					1:
						MEMCPY(ADR(MB_Type), ADR(DstBuf), MIN(MDP_Read.nCount, SIZEOF(MB_Type)) );
						MDP_Read.stMDP_DynAddr.nSubIdx		:= 2;

					2:
						MEMCPY(ADR(SerielNo), ADR(DstBuf), MIN(MDP_Read.nCount, SIZEOF(SerielNo)) );
						MDP_Read.stMDP_DynAddr.nSubIdx		:= 3;

					3:
						MEMCPY(ADR(ProdDate), ADR(DstBuf), MIN(MDP_Read.nCount, SIZEOF(ProdDate)) );
						MDP_Read.stMDP_DynAddr.nSubIdx		:= 4;

					4:
						MEMCPY(ADR(BootCount), ADR(DstBuf), SIZEOF(BootCount));
						MDP_Read.stMDP_DynAddr.nSubIdx		:= 5;

					5:
						MEMCPY(ADR(OpTime), ADR(DstBuf), SIZEOF(OpTime));
						MDP_Read.stMDP_DynAddr.nSubIdx		:= 6;

					6:
						MEMCPY(ADR(MinBoardTemp), ADR(DstBuf), SIZEOF(MinBoardTemp));
						MDP_Read.stMDP_DynAddr.nSubIdx		:= 7;

					7:
						MEMCPY(ADR(MaxBoardTemp), ADR(DstBuf), SIZEOF(MaxBoardTemp));
						MDP_Read.stMDP_DynAddr.nSubIdx		:= 8;

					8:
						MEMCPY(ADR(MinInputVolt), ADR(DstBuf), SIZEOF(MinInputVolt));
						MDP_Read.stMDP_DynAddr.nSubIdx		:= 9;

					9:
						MEMCPY(ADR(MaxInputVolt), ADR(DstBuf), SIZEOF(MaxInputVolt));
						MDP_Read.stMDP_DynAddr.nSubIdx		:= 10;

					10:
						MEMCPY(ADR(MB_Temp), ADR(DstBuf), SIZEOF(MB_Temp));
						MDP_Read.stMDP_DynAddr.nSubIdx		:= 0;
						MDP_Read.stMDP_DynAddr.nTableId		:= 4;
					END_CASE

				4:
					CASE MDP_Read.stMDP_DynAddr.nSubIdx OF
					0:
						MEMCPY(ADR(VoltCount), ADR(DstBuf), SIZEOF(VoltCount) );
						IF VoltCount > 0 THEN
							MDP_Read.stMDP_DynAddr.nSubIdx	:= 1;
						ELSE						
							state							:= 3;
						END_IF

					1..255:
						MEMCPY(ADR(VoltLocation[MDP_Read.stMDP_DynAddr.nSubIdx]), ADR(DstBuf), SIZEOF(VoltLocation[MIN_VOLTAGE]));
						MDP_Read.stMDP_DynAddr.nSubIdx	:= MDP_Read.stMDP_DynAddr.nSubIdx + 1;
						
						IF MDP_Read.stMDP_DynAddr.nSubIdx > VoltCount
						THEN
							MDP_Read.stMDP_DynAddr.nSubIdx	:= 1;
							MDP_Read.stMDP_DynAddr.nTableId	:= 5;
						END_IF
					END_CASE

				5:
					CASE MDP_Read.stMDP_DynAddr.nSubIdx OF
					1..255:
						MEMCPY(ADR(VoltageValue[MDP_Read.stMDP_DynAddr.nSubIdx]), ADR(DstBuf), SIZEOF(VoltageValue[MIN_VOLTAGE]));
						MDP_Read.stMDP_DynAddr.nSubIdx	:= MDP_Read.stMDP_DynAddr.nSubIdx + 1;
						
						IF MDP_Read.stMDP_DynAddr.nSubIdx > VoltCount
						THEN
							MDP_Read.stMDP_DynAddr.nSubIdx	:= 1;
							MDP_Read.stMDP_DynAddr.nTableId	:= 6;
						END_IF
					END_CASE

				6:
					CASE MDP_Read.stMDP_DynAddr.nSubIdx OF
					1..255:
						MEMCPY(ADR(VoltageNominal[MDP_Read.stMDP_DynAddr.nSubIdx]), ADR(DstBuf), SIZEOF(VoltageNominal[MIN_VOLTAGE]));
						MDP_Read.stMDP_DynAddr.nSubIdx	:= MDP_Read.stMDP_DynAddr.nSubIdx + 1;
						
						IF MDP_Read.stMDP_DynAddr.nSubIdx > VoltCount
						THEN
							state							:= 3;
						END_IF
					END_CASE
				END_CASE

				MDP_Read(
					stMDP_DynAddr	:= ,		(* address to request subindex Count of AdressList *)
					pDstBuf			:= ADR(DstBuf),
					cbDstBufLen		:= SIZEOF(DstBuf),
					bExecute		:= NOT MDP_Read.bBusy AND state = 2,
					tTimeout		:= Timeout,
					sAmsNetId		:= AmsNetId,
					bBusy			=> ,
					bError			=> ,
					nErrId			=> );
			END_IF
		END_IF

	3: //Start lesen der IPC Seriennummer 
		MDP_Read.stMDP_DynAddr.nArea						:= INT_TO_BYTE(eMDP_Area_DeviceArea);
		MDP_Read.stMDP_DynAddr.nModuleId					:= 16#9F;
		MDP_Read.stMDP_DynAddr.nTableId						:= 16#00;
		MDP_Read.stMDP_DynAddr.nSubIdx						:= 16#00;
		
		MDP_Read(
			stMDP_DynAddr	:= ,		(* address to request subindex Count of AdressList *)
			pDstBuf			:= ADR(IPC_SerielNo),
			cbDstBufLen		:= SIZEOF(IPC_SerielNo),
			bExecute		:= NOT MDP_Read.bBusy,
			tTimeout		:= Timeout,
			sAmsNetId		:= AmsNetId,
			bBusy			=> ,
			bError			=> ,
			nErrId			=> );	
			
		state												:= 4;	
	
	4:
		MDP_Read( pDstBuf	:= ADR(IPC_SerielNo), cbDstBufLen := SIZEOF(IPC_SerielNo));
		IF NOT MDP_Read.bBusy
		THEN
			IF MDP_Read.bError AND MDP_Read.bExecute
			THEN
				Busy										:= FALSE;
				Error										:= TRUE;
				SplitErrorId(
					nErrID		:= MDP_Read.nErrID,
					eErrGroup	=> ErrorGrp ,
					nErrCode	=> ErrorId);
				state										:= 99;	
			ELSE			                        		
				Busy										:= FALSE;
				Done										:= TRUE;
				state										:= 99;
			END_IF
			MDP_Read(bExecute := FALSE);
			
		END_IF

	99: ;

	ELSE
		;
	END_CASE


	(* reset state for next start *)
	IF NOT Execute
		AND state = 99
	THEN
		state												:= 0;
	END_IF

(****************************************************************************************************)

END_FUNCTION_BLOCK

// POUs/IpcDiag/MDP/InfoModuls/MDP_RaidSimple
{attribute 'no_check'}
FUNCTION_BLOCK MDP_RaidSimple  EXTENDS FbBase
VAR_OUTPUT CONSTANT
	MIN_DRIVE												:	INT := 1;
	MAX_DRIVE												:	INT := 4;
	                    									
//Cntr state            									
	CS_UNKNOWN												:	INT := 0;
	CS_GOOD													:	INT := 1;
	CS_FAILED												:	INT := 2; 
	CS_OFFLINE												:	INT := 3; 
	CS_POWER_OFF											:	INT := 4;
	                    									
//Cntr offline reason   									
	COR_NO_REASON											:	INT := 0;
	COR_INITIALIZING										:	INT := 1;
	COR_BUS_DEGRADED										:	INT := 2;
	COR_BUS_FAILURE											:	INT := 3;
	                    									
//Set state             									
	SS_OK													:	INT := 0;
	SS_DEGRADED												:	INT := 1;
	SS_REBUILDING											:	INT := 2;
	SS_FAILED												:	INT := 3;
	                    									
//Drive state		    									
	DS_OK													:	INT := 0;
	DS_REBUILDING											:	INT := 1;
	DS_FAILED 												:	INT := 2;
	DS_DEGRADED 											:	INT := 3;
END_VAR                 									
VAR_INPUT               									
	AmsNetId												: 	T_AmsNetId := '';	//AmsNetId as text
	Timeout													:	TIME := DEFAULT_ADS_TIMEOUT;	//Ads timeout
END_VAR                 									
VAR_OUTPUT              									
(* Raid Data *)         									
	CntrState												:	INT := CS_UNKNOWN;		//current controller state
	CntrOfflReason 											: 	INT := COR_NO_REASON;	//reason for controller offline
                        									
	SetType													:	USINT;					//type of RAID system
	SetState												:	INT := SS_OK;			
	SetInfo													:	USINT; (* 	If SetStatus = OK, THEN Info will be 0.
																					If SetStatus = DEGRADED, then Info will contain the failed drive index number.1
																					If SetStatus = REBUILDING, then Info will contain the percentage complete. The value will be in the range of 0 to 100 (0h to 64h).
																					If SetStatus == FAILED, then Info will be 0 or vendor specific. Since the failure modes could include drive or controller failures, Info may provide a vendor specific error code to indicate which component led to the failed status. *)
	CountDrives												:	UINT;
	DriveSTATE												:	ARRAY[MIN_DRIVE..MAX_DRIVE] OF INT; //current state of drive
	CountRAIDSets											:	UINT; 		//Count RAID sets
	ErrorGrp												:	E_MDP_ErrGroup := eMDP_Err_NoError;
END_VAR                 									
VAR                     									
	idx														:	INT := 1;
	MDP_ScanModules											:	FB_MDP_ScanModules := ( nModuleType 	:= eMDP_ModT_RAID , iModIdx		:= 0);
	MDP_Read												: 	FB_MDP_Read;
	SplitErrorId											:	FB_MDP_SplitErrorID ;
	DstBuf													:	ARRAY[0..4] OF BYTE;
END_VAR

(* Read RAID Information 						V1.0	*)
(* only for RAID set 1									*)
(* not more then MAX_DRIVES per RAID set				*)
(********************************************************)

(* Start Read *******************************************)
	IF Execute
		AND state = 0
	THEN
		CntrState											:= CS_UNKNOWN;
		CntrOfflReason 										:= COR_NO_REASON;
		SetType												:= 0;
		SetState											:= SS_OK;
		SetInfo												:= 0;
		CountDrives											:= 0;
		MEMSET(ADR(DriveSTATE),0,SIZEOF(DriveSTATE));   	
		CountRAIDSets										:= 0;
                                                        	
		Busy												:= TRUE;
		Done												:= FALSE;
		Error												:= FALSE;
		ErrorId												:= 0;
		ErrorGrp											:= eMDP_Err_NoError;
		MDP_Read(bExecute := FALSE);
		MDP_ScanModules(
			bExecute		:= FALSE,
			nModuleType		:= eMDP_ModT_RAID,
			iModIdx			:= 0,
			tTimeout		:= timeout,
			sAmsNetId		:= AmsNetId,
			bBusy			=> ,
			bError			=> ,
			nErrID			=> ,
			nDynModuleId	=> ,
			iModuleTypeCount=> ,
			iModuleCount	=> );
			
		MDP_ScanModules(bExecute:= TRUE);
		state												:= 1;
	ELSIF NOT Execute
		AND State = 99
	THEN
		state												:= 0;
		Busy												:= FALSE;
		Done												:= FALSE;
		Error												:= FALSE;
		ErrorId												:= 0;
		ErrorGrp											:= eMDP_Err_NoError;
	END_IF


	CASE state OF
	0:
		;
	1:
		MDP_ScanModules();
		IF NOT MDP_ScanModules.bBusy
		THEN
			IF MDP_ScanModules.bError
			THEN
				Busy										:= FALSE;
				Error										:= TRUE;
				SplitErrorId(
					nErrID		:= MDP_ScanModules.nErrID,
					eErrGroup	=> ErrorGrp ,
					nErrCode	=> ErrorId);
				state										:= 99;
				MDP_ScanModules(bExecute := FALSE);
			ELSE
				MDP_Read(bExecute := FALSE);
				MDP_Read.stMDP_DynAddr.nArea				:= 16#8;
				MDP_Read.stMDP_DynAddr.nModuleId			:= MDP_ScanModules.nDynModuleId;
				MDP_Read.stMDP_DynAddr.nTableId				:= 16#1;
				MDP_Read.stMDP_DynAddr.nSubIdx				:= 0;
				state										:= 2;
			END_IF

		END_IF

	2:
		MDP_Read( pDstBuf	:= ADR(DstBuf), cbDstBufLen := SIZEOF(DstBuf));
		IF NOT MDP_Read.bBusy
		THEN
			IF MDP_Read.bError AND MDP_Read.bExecute
			THEN
				IF MDP_Read.stMDP_DynAddr.nTableId = 16#2
					AND MDP_Read.stMDP_DynAddr.nSubIdx = 1
				THEN (* No RaidSystem found *)
					Busy									:= FALSE;
					Done									:= TRUE;
					state									:= 99;
				ELSE
					Busy									:= FALSE;
					Error									:= TRUE;
					SplitErrorId(
						nErrID		:= MDP_Read.nErrID,
						eErrGroup	=> ErrorGrp ,
						nErrCode	=> ErrorId);
				END_IF
				state										:= 99;
				MDP_Read(bExecute := FALSE);
			ELSE
				MDP_Read(bExecute := FALSE);
				CASE MDP_Read.stMDP_DynAddr.nTableId OF
				16#1: (* Controller Info *)
					CASE MDP_Read.stMDP_DynAddr.nSubIdx	OF
					0:
						MDP_Read.stMDP_DynAddr.nSubIdx		:= 1;

					1:
						MEMCPY(ADR(CntrState), ADR(DstBuf), SIZEOF(CntrState));
						MDP_Read.stMDP_DynAddr.nSubIdx		:= 2;

					2:
						MEMCPY(ADR(CntrOfflReason), ADR(DstBuf), SIZEOF(CntrOfflReason));
						MDP_Read.stMDP_DynAddr.nSubIdx		:= 0;
						MDP_Read.stMDP_DynAddr.nTableId		:= 16#2;
					END_CASE

				16#2: (* Raid Sets Type *)
					CASE MDP_Read.stMDP_DynAddr.nSubIdx	OF
					0:
						MEMCPY(ADR(CountRAIDSets), ADR(DstBuf), SIZEOF(CountRAIDSets));
						MDP_Read.stMDP_DynAddr.nSubIdx		:= 1;

					1:
						MEMCPY(ADR(SetType), ADR(DstBuf), SIZEOF(SetType));
						MDP_Read.stMDP_DynAddr.nSubIdx		:= 1;
						MDP_Read.stMDP_DynAddr.nTableId		:= 16#3;
					END_CASE

				16#3: (* RAID sets state and info *)
					CASE MDP_Read.stMDP_DynAddr.nSubIdx	OF
					1:
						MEMCPY(ADR(SetState), ADR(DstBuf[0]), 1);
						MEMCPY(ADR(SetInfo), ADR(DstBuf[1]), 1);
						MDP_Read.stMDP_DynAddr.nSubIdx		:= 0;
						MDP_Read.stMDP_DynAddr.nTableId		:= 16#A;
					END_CASE


				16#A: (* Drives state  *)
					CASE MDP_Read.stMDP_DynAddr.nSubIdx	OF
					0:
						MEMCPY(ADR(CountDrives), ADR(DstBuf), SIZEOF(CountDrives));
						MDP_Read.stMDP_DynAddr.nSubIdx		:= 1;

					1..255:
						MEMCPY(ADR(DriveSTATE), ADR(DstBuf), 1);
						MDP_Read.stMDP_DynAddr.nSubIdx	:= MDP_Read.stMDP_DynAddr.nSubIdx + 1;
						IF MDP_Read.stMDP_DynAddr.nSubIdx > CountDrives
							OR MDP_Read.stMDP_DynAddr.nSubIdx > MAX_DRIVE
						THEN
							Busy							:= FALSE;
							Done							:= TRUE;
							state							:= 99;
						END_IF

					END_CASE

				ELSE
					Busy									:= FALSE;
					Done									:= TRUE;
					state									:= 99;
				END_CASE

				MDP_Read(
					stMDP_DynAddr	:= ,(* address to request subindex Count of AdressList *)
					pDstBuf			:= ADR(DstBuf),
					cbDstBufLen		:= SIZEOF(DstBuf),
					bExecute		:= NOT MDP_Read.bBusy AND state = 2,
					tTimeout		:= Timeout,
					sAmsNetId		:= AmsNetId,
					bBusy			=> ,
					bError			=> ,
					nErrId			=> );
			END_IF
		END_IF

	99: ;

	ELSE
		;
	END_CASE

	(* reset state for next start *)
	IF NOT Execute
		AND state = 99
	THEN
		state												:= 0;
	END_IF

(****************************************************************************************************)

END_FUNCTION_BLOCK

// POUs/IpcDiag/MDP/InfoModuls/MDP_ReadModulList
{attribute 'no_check'}
FUNCTION_BLOCK MDP_ReadModulList EXTENDS FbBase
VAR_INPUT
	AmsNetId												: 	T_AmsNetId := '';	//AmsNetId as text
	Timeout													:	TIME := DEFAULT_ADS_TIMEOUT;	//Ads timeout
END_VAR                     								
VAR_OUTPUT                  								
	ModulCount												:	USINT;	//number of modules
	ModulType												:	ARRAY[0..255] OF E_MDP_ModuleType; //Index = Modul ID
	ErrorGrp												:	E_MDP_ErrGroup := eMDP_Err_NoError;
END_VAR                     								
VAR                         								
	MDP_Read												: 	FB_MDP_Read		:= (stMDP_DynAddr := (nArea := INT_TO_BYTE(eMDP_Area_DeviceArea), nModuleId := 16#02, nTableId := 16#00, nFlag := 16#00, nSubIdx := 16#00));
	SplitErrorId											:	FB_MDP_SplitErrorID;
	dwData													:	ARRAY [1..2] OF WORD;
END_VAR

(* Read list ob available moduls			V1.0	*)
(****************************************************)

(* Start read ************************************************)
	IF Execute
		AND state = 0
	THEN
		IF FALSE
		THEN (* Modultypen Liste *)
			MDP_Read.stMDP_DynAddr.nModuleId				:= 16#01;
		ELSE (* Modul ID Liste *)               			
			MDP_Read.stMDP_DynAddr.nModuleId				:= 16#02;
		END_IF                                  			
		MDP_Read.stMDP_DynAddr.nSubIdx						:= 0;
		MEMSET(ADR(ModulType),0,SIZEOF(ModulType));
		ModulCount											:= 0;
		Busy												:= TRUE;
		Done												:= FALSE;
		Error												:= FALSE;
		ErrorId												:= 0;
		ErrorGrp											:= eMDP_Err_NoError;
		
		MDP_Read(
			stMDP_DynAddr	:= ,		(* address to request subindex Count of AdressList *)
			pDstBuf			:= ADR(dwData),
			cbDstBufLen		:= SIZEOF(dwData),
			bExecute		:= FALSE,
			tTimeout		:= Timeout,
			sAmsNetId		:= AmsNetId,
			bBusy			=> ,
			bError			=> ,
			nErrId			=> );

		MDP_Read(bExecute	:= TRUE);
		state												:= 1;
	ELSIF NOT Execute
		AND State = 99
	THEN
		state												:= 0;
		Busy												:= FALSE;
		Done												:= FALSE;
		Error												:= FALSE;
		ErrorId												:= 0;
		ErrorGrp											:= eMDP_Err_NoError;
	END_IF


	CASE state OF
	0:
		;
	1:
		MDP_Read(pDstBuf := ADR(dwData), cbDstBufLen := SIZEOF(dwData));
		IF NOT MDP_Read.bBusy
		THEN
			IF MDP_Read.bError AND MDP_Read.bExecute
			THEN
				Busy										:= FALSE;
				Error										:= TRUE;
				SplitErrorId(
					nErrID		:= MDP_Read.nErrID,
					eErrGroup	=> ErrorGrp ,
					nErrCode	=> ErrorId);
				state										:= 99;
				MDP_Read(bExecute := FALSE);
			ELSE
				IF ModulCount = 0
				THEN (* Init Modul count *)
					ModulCount								:= WORD_TO_USINT(dwData[1]);
				ELSIF MDP_Read.stMDP_DynAddr.nSubIdx > 0
				THEN (* copy emlement dat					a *)
					ModulType[MDP_Read.stMDP_DynAddr.nSubIdx - 1] :=  dwData[2];					
				END_IF
				MDP_Read(bExecute := FALSE);
				MDP_Read.stMDP_DynAddr.nSubIdx:= MDP_Read.stMDP_DynAddr.nSubIdx + 1;
				IF MDP_Read.stMDP_DynAddr.nSubIdx > ModulCount
					OR MDP_Read.stMDP_DynAddr.nSubIdx > 255
				THEN
					Busy									:= FALSE;
					Done									:= TRUE;
					state									:= 99;
				ELSE
					MDP_Read(bExecute := TRUE,	pDstBuf	:= ADR(dwData), cbDstBufLen := SIZEOF(dwData));
				END_IF
			END_IF

		END_IF

	99: ;

	ELSE
		;
	END_CASE

	(* reset state for next start *)
	IF NOT Execute
		AND state = 99
	THEN
		state												:= 0;
	END_IF

(****************************************************************************************************)

END_FUNCTION_BLOCK

// POUs/IpcDiag/MDP/InfoModuls/MDP_SiliconDrives
{attribute 'no_check'}
FUNCTION_BLOCK MDP_SiliconDrives  EXTENDS FbBase
VAR_OUTPUT CONSTANT
	MIN_DRIVES												:	INT := 1;
	MAX_DRIVES												:	INT := 4;
END_VAR                 									
VAR_INPUT               									
	AmsNetId												: 	T_AmsNetId := '';	//AmsNetId as text
	Timeout													:	TIME := DEFAULT_ADS_TIMEOUT;	//Ads timeout
END_VAR                 									
VAR_OUTPUT              									
	TotEraseCounts											:  ARRAY[MIN_DRIVES..MAX_DRIVES] OF	T_LARGE_INTEGER;	//total number erase operations
	Usage													:	ARRAY[MIN_DRIVES..MAX_DRIVES] OF	UINT;	//usage of drive in %
	NoOfSpares												:	ARRAY[MIN_DRIVES..MAX_DRIVES] OF	UINT;	//number of partitions
	SparedUsed												:	ARRAY[MIN_DRIVES..MAX_DRIVES] OF	UINT;	//usage of partitions
	Count													:	INT; 	//number of drives
	NoSiliconDrives											:	BOOL := FALSE;	//should be TRUE if there is no SSD drive in use
	ErrorGrp												:	E_MDP_ErrGroup := eMDP_Err_NoError;
END_VAR
VAR
	idx														:	INT := 1;
	MDP_ScanModules											:	FB_MDP_ScanModules := ( nModuleType 	:= eMDP_ModT_SiliconDrive , iModIdx		:= 0);
	MDP_Read												: 	FB_MDP_ReadModuleContent;
	SplitErrorId											:	FB_MDP_SplitErrorID;
	DstBuf													:	ARRAY[0..8] OF BYTE;
END_VAR

	(* Read CPU Information 					V1.0	*)
	(****************************************************)

(* Start Read *******************************************************)
	IF Execute
		AND state = 0
	THEN
		MEMSET(ADR(TotEraseCounts),0,SIZEOF(TotEraseCounts));
		MEMSET(ADR(Usage),0,SIZEOF(Usage));
		MEMSET(ADR(NoOfSpares),0,SIZEOF(NoOfSpares));
		MEMSET(ADR(SparedUsed),0,SIZEOF(SparedUsed));
	
		NoSiliconDrives										:= FALSE;
		Count												:= 0;
		Busy												:= TRUE;
		Done												:= FALSE;
		Error												:= FALSE;
		ErrorId												:= 0;
		ErrorGrp											:= eMDP_Err_NoError;
		MDP_Read(bExecute := FALSE);
		MDP_ScanModules(
			bExecute		:= NOT MDP_ScanModules.bExecute,
			nModuleType		:= eMDP_ModT_SiliconDrive,
			iModIdx			:= 0,
			tTimeout		:= timeout,
			sAmsNetId		:= AmsNetId,
			bBusy			=> ,
			bError			=> ,
			nErrID			=> ,
			nDynModuleId	=> ,
			iModuleTypeCount=> ,
			iModuleCount	=> );
		MDP_ScanModules(bExecute := TRUE);
		
		state												:= 1;
	ELSIF NOT Execute
		AND State = 99
	THEN
		state												:= 0;
		Busy												:= FALSE;
		Done												:= FALSE;
		Error												:= FALSE;
		ErrorId												:= 0;
		ErrorGrp											:= eMDP_Err_NoError;
	END_IF


	CASE state OF
	0:
		;
	1:
		MDP_ScanModules();
		IF NOT MDP_ScanModules.bBusy
		THEN
			IF MDP_ScanModules.bError
			THEN
				IF MDP_ScanModules.nErrID = 16#EC800002
				THEN
					Busy									:= FALSE;
					Done									:= TRUE;
					NoSiliconDrives							:= TRUE;
				ELSE

					Busy									:= FALSE;
					Error									:= TRUE;
					SplitErrorId(
						nErrID		:= MDP_ScanModules.nErrID,
						eErrGroup	=> ErrorGrp ,
						nErrCode	=> ErrorId);
				END_IF
				state										:= 99;
				MDP_ScanModules(bExecute := FALSE);
			ELSE
				Count										:= MDP_ScanModules.iModuleTypeCount;
				MDP_Read.stMDP_DynAddr.nArea				:= 16#8;
				MDP_Read.stMDP_DynAddr.nModuleId			:= MDP_ScanModules.nDynModuleId;
				MDP_Read.stMDP_DynAddr.nSubIdx				:= 0;
				MDP_Read.stMDP_DynAddr.nTableId				:= 1;
				MDP_Read(bExecute := FALSE);
				idx											:= 1;
				
				IF Count <= 0
				THEN
					Busy									:= FALSE;
					Done									:= TRUE;
					state									:= 99;
				ELSE
					state									:= 2;
				END_IF
			END_IF

		END_IF

	2:
		MDP_Read( pDstBuf:= ADR(DstBuf), cbDstBufLen:= SIZEOF(DstBuf));
		IF NOT MDP_Read.bBusy
		THEN
			IF MDP_Read.bError AND MDP_Read.bExecute
			THEN
				Busy										:= FALSE;
				Error										:= TRUE;
				SplitErrorId(
					nErrID		:= MDP_Read.nErrID,
					eErrGroup	=> ErrorGrp ,
					nErrCode	=> ErrorId);
				state										:= 99;
				MDP_Read(bExecute := FALSE);
			ELSE
				MDP_Read(bExecute := FALSE);
				CASE MDP_Read.stMDP_DynAddr.nSubIdx OF
				0:
					MDP_Read.stMDP_DynAddr.nSubIdx			:= 1;

				1:
					MEMCPY(ADR(TotEraseCounts[idx]), ADR(DstBuf), MIN(MDP_Read.nCount, SIZEOF(TotEraseCounts[MIN_DRIVES])));
					MDP_Read.stMDP_DynAddr.nSubIdx			:= 2;

				2:
					MEMCPY(ADR(Usage[idx]), ADR(DstBuf), SIZEOF(Usage[MIN_DRIVES]));
					MDP_Read.stMDP_DynAddr.nSubIdx			:= 3;

				3:
					MEMCPY(ADR(NoOfSpares[idx]), ADR(DstBuf), SIZEOF(NoOfSpares[MIN_DRIVES]));
					MDP_Read.stMDP_DynAddr.nSubIdx			:= 4;

				4:
					MEMCPY(ADR(SparedUsed[idx]), ADR(DstBuf), SIZEOF(SparedUsed[MIN_DRIVES]));
					MDP_Read.stMDP_DynAddr.nModuleId		:= MDP_Read.stMDP_DynAddr.nModuleId + 1;
					idx										:= idx + 1;
					MDP_Read.stMDP_DynAddr.nSubIdx			:= 1;
					IF idx > Count
						OR idx > MAX_DRIVES
					THEN
						Busy								:= FALSE;
						Done								:= TRUE;
						state								:= 99;
					END_IF
				END_CASE

				MDP_Read(
					stMDP_DynAddr	:= ,		(* address to request subindex Count of AdressList *)
					pDstBuf			:= ADR(DstBuf),
					cbDstBufLen		:= SIZEOF(DstBuf),
					bExecute		:= NOT MDP_Read.bBusy AND state = 2,
					tTimeout		:= Timeout,
					sAmsNetId		:= AmsNetId,
					bBusy			=> ,
					bError			=> ,
					nErrId			=> );

			END_IF
		END_IF

	99: ;

	ELSE
		;
	END_CASE

	(* reset state for next start *)
	IF NOT Execute
		AND state = 99
	THEN
		state												:= 0;
	END_IF

(****************************************************************************************************)

END_FUNCTION_BLOCK

// POUs/IpcDiag/MDP/InfoModuls/MDP_UPS
{attribute 'no_check'}
FUNCTION_BLOCK MDP_UPS EXTENDS FbBase
VAR_OUTPUT CONSTANT
(* Battery Power Status *)
	PS_UNKNOWN												:	INT := 0;
	PS_ONLINE												:	INT := 1;
	PS_ONBATTERIES											:	INT := 2;
	                    									
(* Com Status *)        									
	CS_UNKNOWN												:	INT := 0;
	CS_OK													:	INT := 1;
	CS_ERROR												:	INT := 2;

(* Battery Power Status *)
	BS_UNKNOWN												:	INT := 0;
	BS_OK													:	INT := 1;
	BS_CHANGE_BATTERY										:	INT := 2;
	
END_VAR
VAR_INPUT
	AmsNetId												: 	T_AmsNetId := '';	//AmsNetId
	Timeout													:	TIME := DEFAULT_ADS_TIMEOUT;	//Ads timeout
END_VAR
VAR_OUTPUT
(* UPS Data *)              								
	Model													:	STRING(30);	//model name
	VendorName												:	STRING(30);	//vendor name
	PowerStatus												:	INT := PS_UNKNOWN;
	ComStatus												:	INT := CS_UNKNOWN;
	BatteryStatus											:	INT := BS_UNKNOWN;
	BatteryCapacity											:	USINT; 		//in %
	BatteryRuntime											:	UDINT; 		//in sec
	PersPowerFailCounter									:	BOOL;		//TRUE when persistent power fail counter is activated
	PowerFailCounter										:	UDINT;		//number of power fails
	FanError												:	BOOL;		//Fan has error
	NoBattery												:	BOOL;		//No battery connected
	ErrorGrp												:	E_MDP_ErrGroup := eMDP_Err_NoError;

END_VAR                     								
VAR                         								
	idx														:	INT := 1;
	MDP_ScanModules											:	FB_MDP_ScanModules := ( nModuleType 	:= eMDP_ModT_UPS , iModIdx		:= 0);
	MDP_Read												: 	FB_MDP_Read;
	SplitErrorId											:	FB_MDP_SplitErrorID;
	DstBuf													:	ARRAY[0..31] OF BYTE;
END_VAR

	(* Read UPS Information 							V1.0	*)
	(***************************************************)

(* Start Read *******************************************************)
	IF Execute
		AND state = 0
	THEN
		Model												:= '';
		VendorName											:= '';
		PowerStatus											:= PS_UNKNOWN;
		ComStatus											:=	CS_UNKNOWN;
		BatteryStatus										:=	BS_UNKNOWN;
		BatteryCapacity										:= 0;
		BatteryRuntime										:= 0;
		PowerFailCounter									:= 0;
		PersPowerFailCounter								:= FALSE;
		FanError											:= FALSE;
		NoBattery											:= FALSE;
		Busy												:= TRUE;
		Done												:= FALSE;
		Error												:= FALSE;
		ErrorId												:= 0;
		ErrorGrp											:= eMDP_Err_NoError;
		MDP_Read(bExecute := FALSE);
		MDP_ScanModules(
			bExecute		:= NOT MDP_ScanModules.bExecute,
			nModuleType		:= eMDP_ModT_UPS,
			iModIdx			:= 0,
			tTimeout		:= timeout,
			sAmsNetId		:= AmsNetId,
			bBusy			=> ,
			bError			=> ,
			nErrID			=> ,
			nDynModuleId	=> ,
			iModuleTypeCount=> ,
			iModuleCount	=> );
			
		MDP_ScanModules(bExecute := TRUE);
		
		state												:= 1;
	ELSIF NOT Execute
		AND State = 99
	THEN
		state												:= 0;
		Busy												:= FALSE;
		Done												:= FALSE;
		Error												:= FALSE;
		ErrorId												:= 0;
		ErrorGrp											:= eMDP_Err_NoError;
	END_IF


	CASE state OF
	0:
		;
	1:
		MDP_ScanModules();
		IF NOT MDP_ScanModules.bBusy
		THEN
			IF MDP_ScanModules.bError
			THEN
				Busy										:= FALSE;
				Error										:= TRUE;
				SplitErrorId(
					nErrID		:= MDP_ScanModules.nErrID,
					eErrGroup	=> ErrorGrp ,
					nErrCode	=> ErrorId);
				state										:= 99;
				MDP_ScanModules(bExecute := FALSE);
			ELSE
				MDP_Read(bExecute := FALSE);
				MDP_Read.stMDP_DynAddr.nArea				:= 16#8;
				MDP_Read.stMDP_DynAddr.nModuleId			:= MDP_ScanModules.nDynModuleId;
				MDP_Read.stMDP_DynAddr.nTableId				:= 1;
				MDP_Read.stMDP_DynAddr.nSubIdx				:= 0;
				state										:= 2;
			END_IF

		END_IF

	2:
		MDP_Read( pDstBuf	:= ADR(DstBuf), cbDstBufLen := SIZEOF(DstBuf));
		IF NOT MDP_Read.bBusy
		THEN
			IF MDP_Read.bError AND MDP_Read.bExecute
			THEN
				Busy										:= FALSE;
				Error										:= TRUE;
				SplitErrorId(
					nErrID		:= MDP_Read.nErrID,
					eErrGroup	=> ErrorGrp ,
					nErrCode	=> ErrorId);
				state										:= 99;
				MDP_Read(bExecute := FALSE);
			ELSE
				MDP_Read(bExecute := FALSE);
				CASE MDP_Read.stMDP_DynAddr.nSubIdx	OF
				0:
					MDP_Read.stMDP_DynAddr.nSubIdx			:= 1;

				1:
					MEMCPY(ADR(Model), ADR(DstBuf), SIZEOF(Model) - 1);
					MDP_Read.stMDP_DynAddr.nSubIdx			:= 2;

				2:
					MEMCPY(ADR(VendorName), ADR(DstBuf), SIZEOF(VendorName) - 1);
					MDP_Read.stMDP_DynAddr.nSubIdx			:= 7;

				7:
					MEMCPY(ADR(PowerStatus), ADR(DstBuf), 1);
					MDP_Read.stMDP_DynAddr.nSubIdx			:= 8;

				8:
					MEMCPY(ADR(ComStatus), ADR(DstBuf), 1);
					MDP_Read.stMDP_DynAddr.nSubIdx			:= 9;

				9:
					MEMCPY(ADR(BatteryStatus), ADR(DstBuf), 1);
					MDP_Read.stMDP_DynAddr.nSubIdx			:= 10;

				10:
					MEMCPY(ADR(BatteryCapacity), ADR(DstBuf), SIZEOF(BatteryCapacity));
					MDP_Read.stMDP_DynAddr.nSubIdx			:= 11;

				11:
					MEMCPY(ADR(BatteryRuntime), ADR(DstBuf), SIZEOF(BatteryRuntime));
					MDP_Read.stMDP_DynAddr.nSubIdx			:= 12;

				12:
					MEMCPY(ADR(PersPowerFailCounter), ADR(DstBuf), SIZEOF(PersPowerFailCounter));
					MDP_Read.stMDP_DynAddr.nSubIdx			:= 13;

				13:
					MEMCPY(ADR(PowerFailCounter), ADR(DstBuf), SIZEOF(PowerFailCounter));
					MDP_Read.stMDP_DynAddr.nSubIdx			:= 14;

				14:
					MEMCPY(ADR(FanError), ADR(DstBuf), SIZEOF(FanError));
					MDP_Read.stMDP_DynAddr.nSubIdx			:= 15;

				15:
					MEMCPY(ADR(NoBattery), ADR(DstBuf), SIZEOF(NoBattery));
					Busy									:= FALSE;
					Done									:= TRUE;
					state									:= 99;
                                                        	
				ELSE                                    	
					Busy									:= FALSE;
					Done									:= TRUE;
					state									:= 99;
				END_CASE

				MDP_Read(
					stMDP_DynAddr	:= ,(* address to request subindex Count of AdressList *)
					pDstBuf			:= ADR(DstBuf),
					cbDstBufLen		:= SIZEOF(DstBuf),
					bExecute		:= NOT MDP_Read.bBusy AND state = 2,
					tTimeout		:= Timeout,
					sAmsNetId		:= AmsNetId,
					bBusy			=> ,
					bError			=> ,
					nErrId			=> );
			END_IF
		END_IF

	99: ;

	ELSE
		;
	END_CASE

	(* reset state for next start *)
	IF NOT Execute
		AND state = 99
	THEN
		state												:= 0;
	END_IF

(****************************************************************************************************)

END_FUNCTION_BLOCK

// POUs/IpcDiag/MDP/MDP_Info
{attribute 'no_check'}
//Wrapper for available MDP_xxxx FBs of the lib, based on Beckhoff MDP - invalid values are reported via EventLogger 
//based on Tc2_MDP.lib - please see Beckhoff documentation for further information about Tc2_MDP.lib (IPC diagnostics)
FUNCTION_BLOCK MDP_Info EXTENDS FbBase
VAR_OUTPUT CONSTANT
	FNC_READ_ALL											:	INT := 0;
	FNC_READ_MOD_LIST										:	INT := 1;
	FNC_READ_MB												:	INT := 2;
	FNC_READ_CPU											:	INT := 3;
	FNC_READ_FAN											:	INT := 4;
	FNC_READ_SD												:	INT := 5;
	FNC_READ_RAID											:	INT := 6;
	FNC_READ_UPS											:	INT := 7;
END_VAR                 									
VAR_INPUT               									
	AmsNetId												: 	T_AmsNetId := '';	//AmsNetId as text
	Timeout													:	TIME := DEFAULT_ADS_TIMEOUT; //Ads timeout
	Fnc														:	INT (FNC_READ_ALL..FNC_READ_UPS) := FNC_READ_ALL; //select function to be read
(* Components *)            								
	ModList													:	MDP_ReadModulList;	//see content in FB
	MB														:	MDP_Mainboard;		//see content in FB
	CPU														:	MDP_CPU;			//see content in FB
	FAN														:	MDP_Fan;			//see content in FB
	SD														:	MDP_SiliconDrives;	//see content in FB
	RAID													:	MDP_RaidSimple;		//see content in FB
	UPS														:	MDP_UPS;			//see content in FB
END_VAR                     								
VAR_OUTPUT                  								
	TotalCycleTime											:	TIME;	//Cylce time to execute function block with mode read all        
	ErrorGrp												:	E_MDP_ErrGroup;
	ErrorFnc												:	STRING(15);
END_VAR
VAR
	MemFnc													:	INT;
	MemExecute												:	BOOL;
	MemErrorFnc												:	STRING(15);
	MemErrorid												:	UDINT;
	MemErrorGrp												:	E_MDP_ErrGroup;
	MemTimeStartCycle										:	TIME;
END_VAR

	(* Execute all available MDP_xxxxx fb 			*)
	(************************************************)

(* Sequence ********************************************)
	IF Execute
		AND state = 0
	THEN
		ReadAll(Execute	:= Execute);
	ELSIF state <> 0
	THEN
		ReadAll(Execute	:= Execute);
	END_IF

(*****************************************************************************)

METHOD PUBLIC readAll : BOOL //Return value = TRUE if busy;
VAR_INPUT
	Execute													:	BOOL;
END_VAR
	THIS^.Execute											:= Execute;

	IF Execute
		AND State = 0
	THEN
		MemFnc												:= Fnc;
		CASE Fnc OF                                     	
		FNC_READ_MOD_LIST:		state						:= 10;
		FNC_READ_MB:			state						:= 20;
		FNC_READ_CPU:			state						:= 30;
		FNC_READ_FAN:			state						:= 40;
		FNC_READ_SD:			state						:= 50;
		FNC_READ_RAID:	 		state						:= 60;
		FNC_READ_UPS:	 		state						:= 70;
		ELSE (* Read All *)
			MemFnc											:= FNC_READ_ALL;
			state											:= 10;
		END_CASE
		MemTimeStartCycle									:= TIME();
		Busy												:= TRUE;
		Done												:= FALSE;
		Error												:= FALSE;
		Errorid												:= 0;
		ErrorFnc											:= '';
		ErrorGrp											:= eMDP_Err_NoError;
		MemExecute											:= FALSE;
		MemErrorid											:= 0;
		MemErrorFnc											:= '';
		MemErrorGrp											:= eMDP_Err_NoError;
	ELSIF NOT Execute
		AND State = 99
	THEN
		Busy												:= FALSE;
		Done												:= FALSE;
		Error												:= FALSE;
		Errorid												:= 0;
		ErrorFnc											:= '';
		ErrorGrp											:= eMDP_Err_NoError;
		MemExecute											:= FALSE;
		MemErrorid											:= 0;
		MemErrorFnc											:= '';
		MemErrorGrp											:= eMDP_Err_NoError;
		ReadModList(FALSE);     						
		ReadMB(FALSE);
		ReadCPU(FALSE);
		ReadFAN(FALSE);
		ReadSD(FALSE);
		ReadRaid(FALSE);
	END_IF

	CASE state OF
	10:

		MemExecute											:= TRUE;
		ReadModList(MemExecute);
		IF NOT ModList.Busy
		THEN
			IF MemFnc = FNC_READ_ALL
			THEN
				IF Error AND MemErrorid = 0 
				THEN
					MemErrorId								:= Errorid; 
					MemErrorFnc 							:= CONCAT('ReadModList Fnc:',TO_STRING(FNC_READ_MOD_LIST)); 
					MemErrorGrp 							:= ErrorGrp;
				END_IF              						
				Busy										:= TRUE;
				Done										:= FALSE;
				Error										:= FALSE;
				Errorid										:= 0;
				ErrorGrp									:= eMDP_Err_NoError;
				state										:= 20;
			ELSE                    						
				state										:= 99;
			END_IF
		END_IF

	20:
		MemExecute											:= TRUE;
		ReadMB(MemExecute);
		IF NOT MB.Busy
		THEN
			IF MemFnc = FNC_READ_ALL
			THEN
				IF Error AND MemErrorid = 0 
				THEN
					MemErrorId								:= Errorid; 
					MemErrorFnc 							:= CONCAT('ReadMB Fnc: ',TO_STRING(FNC_READ_MB));  
					MemErrorGrp 							:= ErrorGrp;
				END_IF              						
				Busy										:= TRUE;
				Done										:= FALSE;
				Error										:= FALSE;
				Errorid										:= 0;
				ErrorGrp									:= eMDP_Err_NoError;
				state										:= 30;
			ELSE                    						
				state										:= 99;
			END_IF                  	
		END_IF

	30:
		MemExecute											:= TRUE;
		ReadCPU(MemExecute);
		IF NOT CPU.Busy
		THEN
			IF MemFnc = FNC_READ_ALL
			THEN
				IF Error AND MemErrorid = 0 THEN
					MemErrorId								:= Errorid; 
					MemErrorFnc 							:= CONCAT('ReadCPU Fnc: ',TO_STRING(FNC_READ_CPU));  
					MemErrorGrp 							:= ErrorGrp;
				END_IF              						
				Busy										:= TRUE;
				Done										:= FALSE;
				Error										:= FALSE;
				Errorid										:= 0;
				ErrorGrp									:= eMDP_Err_NoError;
				state										:= 40;
			ELSE                    						
				state										:= 99;
			END_IF
		END_IF

	40:
		MemExecute											:= TRUE;
		ReadFan(MemExecute);
		IF NOT Fan.Busy
		THEN
			IF MemFnc = FNC_READ_ALL
			THEN
				IF Error AND MemErrorid = 0 
				THEN
					MemErrorId								:= Errorid; 
					MemErrorFnc 							:= CONCAT('ReadFan Fnc: ',TO_STRING(FNC_READ_FAN));  
					MemErrorGrp 							:= ErrorGrp;
				END_IF              						
				Busy										:= TRUE;
				Done										:= FALSE;
				Error										:= FALSE;
				Errorid										:= 0;
				ErrorGrp									:= eMDP_Err_NoError;
				state										:= 50;
			ELSE                    						
				state										:= 99;
			END_IF
		END_IF

	50:
		MemExecute											:= TRUE;		
		ReadSD(MemExecute);
		
		IF NOT SD.Busy
		THEN
			IF MemFnc = FNC_READ_ALL
			THEN
				IF Error AND MemErrorid = 0 
				THEN				
					MemErrorId								:= Errorid; 
					MemErrorFnc 							:= CONCAT('ReadSD Fnc: ',TO_STRING(FNC_READ_SD)); 
					MemErrorGrp 							:= ErrorGrp;
				END_IF              						
				Busy										:= TRUE;
				Done										:= FALSE;
				Error										:= FALSE;
				Errorid										:= 0;
				ErrorGrp									:= eMDP_Err_NoError;
				state										:= 60;
			ELSE                    						
				state										:= 99;
			END_IF                  	
		END_IF

	60:
		MemExecute											:= TRUE;
		ReadRaid(MemExecute);
		IF NOT Raid.Busy
		THEN
			IF MemFnc = FNC_READ_ALL
			THEN
				IF Error AND MemErrorid = 0 
				THEN
					MemErrorId								:= Errorid; 
					MemErrorFnc 							:= CONCAT('ReadRaid Fnc: ',TO_STRING(FNC_READ_RAID));
					MemErrorGrp 							:= ErrorGrp;
				END_IF              						
				Busy										:= TRUE;
				Done										:= FALSE;
				Error										:= FALSE;
				Errorid										:= 0;
				ErrorGrp									:= eMDP_Err_NoError;
				state										:= 70;
			ELSE                    						
				state										:= 99;
			END_IF
		END_IF

	70:
		MemExecute											:= TRUE;
		ReadUPS(MemExecute);
		IF NOT UPS.Busy
		THEN
			IF TRUE
			THEN
				IF Error AND MemErrorid = 0 
				THEN
					MemErrorId								:= Errorid; 
					MemErrorFnc 							:= CONCAT('ReadUPS Fnc: ',TO_STRING(FNC_READ_UPS));
					MemErrorGrp 							:= ErrorGrp;
				END_IF
				Busy										:= FALSE;
				Done										:= MemErrorId = 0;
				Error										:= MemErrorId <> 0;
				Errorid										:= MemErrorid;
				ErrorFnc									:= MemErrorFnc;
				ErrorGrp									:= MemErrorGrp;
				state										:= 99;
			ELSE                    						
				state										:= 99;
			END_IF
		END_IF

	99:;
	
	END_CASE

	IF state = 99
	THEN
		TotalCycleTime	 									:= TIME() - MemTimeStartCycle;
		IF NOT Execute
		THEN
			state											:= 0;
			ReadModList(FALSE);         					
			ReadMB(FALSE);              					
			ReadCPU(FALSE);             					
			ReadFAN(FALSE);             					
			ReadSD(FALSE);              					
			ReadRaid(FALSE);            					
			ReadUPS(FALSE);             	
		END_IF                          	
	END_IF                              	
	                                    	
	ReadAll													:= Busy;

(***********************************************************************************)
END_METHOD

METHOD PUBLIC readCPU : BOOL //Return value = TRUE if busy
VAR_INPUT
	Execute													:	BOOL;
END_VAR
THIS^.Execute												:= Execute;

CPU(
	Execute				:= MemExecute OR Execute,
	AmsNetId			:= AmsNetId,
	Timeout				:= Timeout,
	MIN_CPU				=> ,
	MAX_CPU				=> ,
	Busy				=> Busy,
	Done				=> Done,
	Error				=> Error,
	ErrorId				=> Errorid,
	ErrorGrp 			=> ErrorGrp,
	Frequency			=> ,
	Usage				=> ,
	Temperature			=> ,
	AverageFrequency	=> ,
	AverageUsage		=> ,
	AverageTemperature	=> ,
	Count				=> );

MemExecute 													:= FALSE;
	        												
ReadCPU														:= Busy;
END_METHOD

METHOD PUBLIC readFan : BOOL //Return value = TRUE if busy
VAR_INPUT
	Execute													:	BOOL;
END_VAR
THIS^.Execute												:= Execute;

FAN(
	Execute		:= MemExecute OR Execute,
	AmsNetId	:= AmsNetid,
	Timeout		:= Timeout,
	MIN_FAN		=> ,
	MAX_FAN		=> ,
	Busy		=> Busy,
	Done		=> Done,
	Error		=> Error,
	ErrorId		=> ErrorId,
	ErrorGrp 	=> ErrorGrp,
	Speed		=> ,
	Count		=> );

MemExecute 													:= FALSE;
           												
ReadFan														:= Busy;
END_METHOD

METHOD PUBLIC readMB : BOOL //Return value = TRUE if busy
VAR_INPUT
	Execute													:	BOOL;
END_VAR
THIS^.Execute												:= Execute;

MB(
	Execute			:= MemExecute OR Execute,
	AmsNetId		:= AmsNetId,
	Timeout			:= Timeout,
	MIN_VOLTAGE		=> ,
	MAX_VOLTAGE		=> ,
	Busy			=> Busy,
	Done			=> Done,
	Error			=> Error,
	ErrorId			=> ErrorId,
	ErrorGrp		=> Errorgrp,
	MB_Type			=> ,
	SerielNo		=> ,
	ProdDate		=> ,
	BootCount		=> ,
	OpTime			=> ,
	MinBoardTemp	=> ,
	MaxBoardTemp	=> ,
	MinInputVolt	=> ,
	MaxInputVolt	=> ,
	MB_Temp			=> ,
	VoltLocation	=> ,
	VoltageValue	=> ,
	VoltageNominal	=> ,
	VoltCount		=> );

MemExecute 													:= FALSE;
            												
ReadMB														:= Busy;
END_METHOD

METHOD PUBLIC readModList : BOOL //Return value = TRUE if busy
VAR_INPUT
	Execute													:	BOOL;
END_VAR
THIS^.Execute												:= Execute;

ModList(
	Execute		:= MemExecute OR Execute,
	AmsNetId	:= AmsNetId,
	Timeout		:= Timeout,
	Busy		=> Busy,
	Done		=> done,
	Error		=> Error,
	ErrorId		=> ErrorId,
	ErrorGrp 	=> ErrorGrp );

MemExecute 													:= FALSE;
            												
ReadModList													:= Busy;
END_METHOD

METHOD PUBLIC readRaid : BOOL //Return value = TRUE if busy
VAR_INPUT
	Execute													: BOOL;
END_VAR
THIS^.Execute												:= Execute;

RAID(
	Execute			:= Execute OR MemExecute,
	AmsNetId		:= AmsNetId,
	Timeout			:= timeout,
	MIN_DRIVE		=> ,
	MAX_DRIVE		=> ,
	Busy			=> Busy,
	Done			=> done,
	Error			=> Error,
	ErrorId			=> ErrorId,
	ErrorGrp 		=> ErrorGrp,
	CntrState		=> ,
	CntrOfflReason	=> ,
	SetType			=> ,
	SetState		=> ,
	SetInfo			=> ,
	CountDrives		=> ,
	DriveSTATE		=> ,
	CountRAIDSets	=> );

MemExecute 													:= FALSE;
                											
ReadRaid													:= Busy;
END_METHOD

METHOD PUBLIC readSD : BOOL //Return value = TRUE if busy
VAR_INPUT
	Execute		:	BOOL;
END_VAR
THIS^.Execute												:= Execute;

SD(
	Execute			:= MemExecute OR Execute,
	AmsNetId		:= AmsNetid,
	Timeout			:= timeout,
	MIN_DRIVES		=> ,
	MAX_DRIVES		=> ,
	Busy			=> Busy,
	Done			=> Done,
	Error			=> Error,
	ErrorId			=> Errorid,
	ErrorGrp 		=> ErrorGrp,
	TotEraseCounts	=> ,
	Usage			=> ,
	NoOfSpares		=> ,
	SparedUsed		=> ,
	Count			=> );

MemExecute	 												:= FALSE;
                											
ReadSD														:= Busy;
END_METHOD

METHOD PUBLIC readUPS : Bool //Return value = TRUE if busy
VAR_INPUT
	Execute		:	BOOL;
END_VAR
THIS^.Execute												:= Execute;

UPS(
	Execute					:= MemExecute OR Execute,
	AmsNetId				:= AmsNetid,
	Timeout					:= timeout,
	Busy					=> Busy,
	Done					=> Done,
	Error					=> Error,
	ErrorId					=> Errorid,
	ErrorGrp				=> ErrorGrp,
	Model					=> ,
	VendorName				=> ,
	PowerStatus				=> ,
	ComStatus				=> ,
	BatteryStatus			=> ,
	BatteryCapacity			=> ,
	BatteryRuntime			=> ,
	PersPowerFailCounter	=> ,
	PowerFailCounter		=> ,
	FanError				=> ,
	NoBattery				=> );

MemExecute 													:= FALSE;
ReadUPS														:= Busy;
END_METHOD

END_FUNCTION_BLOCK

// POUs/IpcDiag/MDP/MDP_IpcDiag
{attribute 'no_check'}
//General IPC diagnosis based on Beckhoff MDP - invalid values are reported via EventLogger 
//based on Tc2_MDP.lib - please see Beckhoff documentation for further information about Tc2_MDP.lib (IPC diagnostics)
//EventHandlingGrp10 instance used inside
//Info:
// 0x   	a    	nn   	x   
// 0x   	8   	03   	1   
// a 	= Area Code (e.g. 8 = Configuration Area) 
// nn 	= Modul-ID (e.g. dynamic modul id from list F020) 
// x	= Tabel id (e.g. 1 = Table 0x8nn1 - NIC Properties at area code 8) 
FUNCTION_BLOCK MDP_IpcDiag
VAR CONSTANT
	MIN_CPU													:	INT := 1;
	MAX_CPU													:	INT := 4;
	                    									
	MIN_FAN													:	INT := 1;
	MAX_FAN													:	INT := 4;
	                    									
	MIN_VOLTAGE												:	INT := 1;
	MAX_VOLTAGE												:	INT := 8;		
END_VAR                 									
VAR_INPUT               									
	Enable													:	BOOL := FALSE;	//FB will be processed as long as enable is TRUE 
	CycleTime												:	TIME := T#100MS; //Delay between ads call to read a single value 
	AmsNetId												: 	T_AmsNetId := ''; //Ams net Id
	Timeout													: 	TIME := DEFAULT_ADS_TIMEOUT; //Ads timeout
{attribute 'displaymode':='bin'}
	FanMask													:	BYTE := 2#0000_0011; //Installed fans inside the PC 
	
//Threshold values 	    									
	MinSpeedFan												:	INT := 2500; 	//rpm
	MaxTempMB												:	INT := 85; 		//°C
	MaxTempCPU												:	INT := 100; 	//°C
	TempWarningThreshold									:	INT := 10; 		//°C
	VoltageFactor											:	LREAL := 0.7; 	//% of nominal voltage before an error occurs
END_VAR                 									
VAR_OUTPUT              										                									
	MB_Temp													:	INT; //Motherboard temp with one decimal digit  
	Voltage_Count											:	INT := 0; //count of voltage measurement points with one decimal digit 
	MB_NominalVoltage										:	ARRAY[MIN_VOLTAGE..MAX_VOLTAGE] OF INT; //in mV
	MB_Voltage												:	ARRAY[MIN_VOLTAGE..MAX_VOLTAGE] OF INT;  //in mV
	CPU_Count												:	INT := 0; //Readed number of CPUs
	CPU_Temp												:	ARRAY[MIN_CPU..MAX_CPU] OF INT; //cpu temperatur with one decimal digit
	FAN_Count												:	INT := 0; //Number of FANs in config. Note, the number may be two where only the second fan is p
	FAN_Speed												:	ARRAY[MIN_FAN..MAX_FAN] OF INT; //in rpm for each available fan
	OsImage													:	STRING; //Image version 
	ExecutionTime											:	TIME; 	//Cylce time to execute function block        
	Busy													:	BOOL;	//Busy is TRUE at the rising edge of Enable and stays TRUE as long as the FB is performing any action. 
	Valid													:	BOOL;	//data valid
	Error													:	BOOL;	//Rising edge of Error informs that an error occurred during the execution of the Function Block 
{attribute 'displaymode':='hex'}
	ErrorId													:	UDINT;	//Error identification - see documentation about IPC diagnostic for further detailed informantion 
	ErrorGrp												:	E_MDP_ErrGroup := eMDP_Err_NoError; //MDP Error code - see Beckhoff documentation MDP for further informantion
END_VAR	
VAR
(* cache variables ************************************************************)
	state													:	INT := 0;
	
	dwData													:	ARRAY [1..2] OF WORD;
	                    									
	MemLen													:	BYTE := 0;
	MemModIdMB												:	BYTE;
	MemModIdCPU												:	ARRAY[MIN_CPU..MAX_CPU] OF BYTE;
	MemModIdFan												:	ARRAY[MIN_FAN..MAX_FAN] OF BYTE;
	MEmModIdUPS												:	BYTE;
	MemMBSubIdxVoltage										:	ARRAY[MIN_VOLTAGE..MAX_VOLTAGE] OF BYTE;
	MemTimeStartCycle										:	TIME;
	MemErrState												:	INT := 0;
	
(* timer ***************************************************************************)
	TON_Cycle												:	TON;
	
(* function-blocks *****************************************************************)
	MDP_Read												: 	FB_MDP_Read		:= (tTimeout := DEFAULT_ADS_TIMEOUT, stMDP_DynAddr := (nArea := INT_TO_BYTE(eMDP_Area_DeviceArea), nModuleId := 16#02, nTableId := 16#00, nFlag := 16#00, nSubIdx := 16#00));
	SplitErrorId											:	FB_MDP_SplitErrorID;
	
(* internal used variables **********************************************************)
	i,k														:	INT;

END_VAR

(* MDP IPC diag compact						V1.1	*)
(****************************************************)

(* Sequence *******************************************************)
IF Enable
THEN
	CASE state OF
	0:	
		IF NOT MDP_Read.bBusy
			AND NOT Error
		THEN
			Busy											:= TRUE;
			Valid											:= FALSE;
		
			Fan_Count										:= 0;
			CPU_Count										:= 0;
			Voltage_Count									:= 0;
			MemLen											:= 0;
			MB_Temp											:= 0;
			MEMSET(ADR(MB_Voltage),0,SIZEOF(MB_Voltage));
			MEMSET(ADR(CPU_Temp),0,SIZEOF(CPU_Temp));
			MEMSET(ADR(FAN_Speed),0,SIZEOF(FAN_Speed));
			MEMSET(ADR(MemModIdCPU),0,SIZEOF(MemModIdCPU));
			MEMSET(ADR(MemModIdFan),0,SIZEOF(MemModIdFan));
			MEMSET(ADR(MemMBSubIdxVoltage),0,SIZEOF(MemMBSubIdxVoltage));
			MEMSET(ADR(MB_NominalVoltage),0,SIZEOF(MB_NominalVoltage));
			
			MDP_Read.stMDP_DynAddr.nArea					:= INT_TO_BYTE(eMDP_Area_GeneralArea);
			MDP_Read.stMDP_DynAddr.nModuleId				:= 16#00;
			MDP_Read.stMDP_DynAddr.nTableId					:= 16#0A;
			MDP_Read.stMDP_DynAddr.nSubIdx					:= 16#00;
                                                    			                                        		
			state											:= 1;
		ELSE
			MDP_Read(bExecute := FALSE);	
		END_IF
		
	1:
	//Read OS version 	
		MDP_Read(bExecute := TRUE , pDstBuf := ADR(OsImage), cbDstBufLen := SIZEOF(OsImage));
		IF NOT MDP_Read.bBusy
		THEN
			IF MDP_Read.bError AND MDP_Read.bExecute
			THEN
				Busy										:= FALSE;
				Error										:= TRUE;
				SplitErrorId(
					nErrID		:= MDP_Read.nErrID,
					eErrGroup	=> ErrorGrp ,
					nErrCode	=> ErrorId);
				MemErrState									:= state;		
				state										:= 99;
				MDP_Read(bExecute := FALSE);
			ELSE //Os Image readed
				k											:= UDINT_TO_INT(MDP_Read.nCount + 1);	
				OsImage[k]									:= 0; //Terminate string
				MDP_Read(bExecute := FALSE);	
				
				//Deveice area F + Modul Id 02 + Tabel Id = 0 -> Index 0xF020 – Modul ID Liste in deveice area
				MDP_Read.stMDP_DynAddr.nArea				:= INT_TO_BYTE(eMDP_Area_DeviceArea); //Index F
				MDP_Read.stMDP_DynAddr.nModuleId			:= 16#02; //Modul id 02 in Config area dynamic modul ids are used!
				MDP_Read.stMDP_DynAddr.nTableId				:= 16#00; //Table Id 0
				MDP_Read.stMDP_DynAddr.nSubIdx				:= 16#00; //Len = number of dyn moduls			
				state										:= 2;								
			END_IF
		END_IF		
		
	2: // search list with dynamic moduls
		MDP_Read(bExecute := TRUE, pDstBuf := ADR(dwData), cbDstBufLen := SIZEOF(dwData));
		IF NOT MDP_Read.bBusy
		THEN
			IF MDP_Read.bError AND MDP_Read.bExecute
			THEN
				Busy										:= FALSE;
				Error										:= TRUE;
				SplitErrorId(
					nErrID		:= MDP_Read.nErrID,
					eErrGroup	=> ErrorGrp ,
					nErrCode	=> ErrorId);
				MemErrState									:= state;	
				state										:= 99;
				MDP_Read(bExecute := FALSE);
			ELSE
				IF MemLen = 0
				THEN (* Init Modul count *)
					MemLen									:= WORD_TO_BYTE(dwData[1]);
				ELSIF MDP_Read.stMDP_DynAddr.nSubIdx > 0
				THEN (* copy emlement dat					a *)
					CASE dwData[2] OF //High word = Modul type, Low word = Modul Id
					Tc2_MDP.E_MDP_ModuleType.eMDP_ModT_Mainboard:
						MemModIdMB		 					:= WORD_TO_BYTE(dwData[1]);		

					Tc2_MDP.E_MDP_ModuleType.eMDP_ModT_UPS:
						MEmModIdUPS							:= WORD_TO_BYTE(dwData[1]);

					Tc2_MDP.E_MDP_ModuleType.eMDP_ModT_CPU:
						CPU_Count							:= CPU_Count + 1;
						MemModIdCPU[CPU_Count]				:= WORD_TO_BYTE(dwData[1]);

					Tc2_MDP.E_MDP_ModuleType.eMDP_ModT_Fan:
						Fan_Count							:= Fan_Count + 1;
						MemModIdFan[Fan_Count]				:= WORD_TO_BYTE(dwData[1]);
												
					ELSE
						; 
					END_CASE				
				END_IF
				MDP_Read(bExecute := FALSE);
				MDP_Read.stMDP_DynAddr.nSubIdx:= MDP_Read.stMDP_DynAddr.nSubIdx + 1;
				IF MDP_Read.stMDP_DynAddr.nSubIdx > MemLen
					OR MDP_Read.stMDP_DynAddr.nSubIdx > 255
				THEN
					state									:= SEL(MemModIdMB > 0 , 9 , 3);								
				ELSE
					MDP_Read(bExecute := TRUE,	pDstBuf	:= ADR(dwData), cbDstBufLen := SIZEOF(dwData));
				END_IF
			END_IF

		END_IF
				
	3: //reading motherboardconfig (SubIndex Voltage)
		MDP_Read.stMDP_DynAddr.nArea						:= INT_TO_BYTE(eMDP_Area_ConfigArea);
		MDP_Read.stMDP_DynAddr.nModuleId					:= INT_TO_BYTE(MemModIdMB);
		MDP_Read.stMDP_DynAddr.nTableId						:= 16#04;
		MDP_Read.stMDP_DynAddr.nSubIdx						:= 16#00;
		MemLen												:= 0;
		i													:= 0;
		
		MDP_Read(
			stMDP_DynAddr	:= ,		(* address to request subindex Count of AdressList *)
			pDstBuf			:= ADR(dwData[1]),
			cbDstBufLen		:= SIZEOF(dwData[1]),
			bExecute		:= NOT MDP_Read.bBusy,
			tTimeout		:= ,
			sAmsNetId		:= AmsNetId,
			bBusy			=> ,
			bError			=> ,
			nErrId			=> );	
			
		state												:= 4;	
	
	4: 
		MDP_Read(pDstBuf := ADR(dwData[1]), cbDstBufLen := SIZEOF(dwData[1]));
		IF NOT MDP_Read.bBusy
		THEN
			IF MDP_Read.bError AND MDP_Read.bExecute
			THEN
				Busy										:= FALSE;
				Error										:= TRUE;
				SplitErrorId(
					nErrID		:= MDP_Read.nErrID,
					eErrGroup	=> ErrorGrp ,
					nErrCode	=> ErrorId);
				MemErrState									:= state;		
				state										:= 99;
				MDP_Read(bExecute := FALSE);
			ELSE
				IF MemLen = 0
				THEN (* Init Entry count *)
					MemLen									:= WORD_TO_BYTE(dwData[1]);
				ELSE 
					MDP_Read(bExecute := FALSE);
					(* copy emlement data
						00 = LOCATION_UNKNOWN
						01 = LOCATION_OTHER
						02 = LOCATION_PROCESSOR
						03 = LOCATION_DISK
						04 = LOCATION_SYSTEM_MANAGEMENT_MODULE
						05 = LOCATION_MOTHERBOARD
						06 = LOCATION_MEMORY_MODULE
						07 = LOCATION_POWER_SUPPLY
						08 = LOCATION_ADDIN_CARD
						09 = LOCATION_FRONT_PANEL_BOARD
						10 = LOCATION_BACK_PANEL_BOARD
						11 = LOCATION_PERIPHERIE
						12 = LOCATION_CHASSIS
						13 = LOCATION_BATTERY
						14 = LOCATION_UPS
						15 = LOCATION_GRAFFIC_BOARD
						16 = LOCATION_SUPERIO
						17 = LOCATION_CHIPSET
					*)

				
					CASE dwData[1] OF
					7, //PowerSupply			
					13: //Battery
						Voltage_Count						:= Voltage_Count + 1;
						MemMBSubIdxVoltage[Voltage_Count]	:= MDP_Read.stMDP_DynAddr.nSubIdx; 
					ELSE
						; 
					END_CASE			
					MDP_Read.stMDP_DynAddr.nSubIdx			:= MDP_Read.stMDP_DynAddr.nSubIdx + 1; 				
							
					IF MDP_Read.stMDP_DynAddr.nSubIdx > MemLen
						OR MDP_Read.stMDP_DynAddr.nSubIdx > 255
						OR Voltage_Count >= MAX_Voltage
					THEN
						IF Voltage_Count > 0
						THEN
							i 								:= MIN_VOLTAGE;
							MDP_Read.stMDP_DynAddr.nTableId	:= 16#06;
							MDP_Read.stMDP_DynAddr.nSubIdx	:= MemMBSubIdxVoltage[i];
							MDP_Read(bExecute := TRUE,	pDstBuf	:= ADR(dwData[1]), cbDstBufLen := SIZEOF(dwData[1]));												
							state							:= 5;				
						ELSE
							state							:= 9;	
						END_IF
				
					ELSE
						MDP_Read(bExecute := TRUE,	pDstBuf	:= ADR(dwData[1]), cbDstBufLen := SIZEOF(dwData[1]));
					END_IF
				END_IF
			END_IF

		END_IF	

	5:	//Nominal Voltage lesen
		MDP_Read(pDstBuf := ADR(dwData[1]), cbDstBufLen := SIZEOF(dwData[1]));
		IF NOT MDP_Read.bBusy
		THEN
			IF MDP_Read.bError AND MDP_Read.bExecute
			THEN
				Busy										:= FALSE;
				Error										:= TRUE;
				SplitErrorId(
					nErrID		:= MDP_Read.nErrID,
					eErrGroup	=> ErrorGrp ,
					nErrCode	=> ErrorId);
				MemErrState									:= state;		
				state										:= 99;
				MDP_Read(bExecute := FALSE);
			ELSE //Nominal Volage
				MDP_Read(bExecute := FALSE);
				MB_NominalVoltage[i]						:= WORD_TO_INT(dwData[1]); 
				i 											:= i + 1;
				IF i > MAX_VOLTAGE
					OR i > Voltage_Count
				THEN //Ende der Bearbeitung
					state									:= 9;								
				ELSE
					MDP_Read.stMDP_DynAddr.nSubIdx			:= MemMBSubIdxVoltage[i];
					MDP_Read(bExecute := TRUE,	pDstBuf	:= ADR(dwData[1]), cbDstBufLen := SIZEOF(dwData[1]));
				END_IF
			END_IF

		END_IF	
							
	//Start Cylce Read
	9: 	
		TON_Cycle(IN := FALSE);
		MemTimeStartCycle									:= T#0MS;
		i													:= 0;
		state												:= 10;	
		
	//Start lesen der Zyklischen Daten 
	10..90: 
		MDP_Read(pDstBuf := ADR(dwData[1]), cbDstBufLen := SIZEOF(dwData[1]));
		IF NOT MDP_Read.bBusy
		THEN			
			IF MDP_Read.bError AND MDP_Read.bExecute
			THEN
				Busy										:= FALSE;
				Error										:= TRUE;
				SplitErrorId(
					nErrID		:= MDP_Read.nErrID,
					eErrGroup	=> ErrorGrp ,
					nErrCode	=> ErrorId);
				MemErrState									:= state;	
				state										:= 99;
				MDP_Read(bExecute := FALSE);
			ELSIF NOT TON_Cycle.IN
			THEN		
				MDP_Read(bExecute := FALSE);
				CASE state OF
				10:
					MDP_Read.stMDP_DynAddr.nModuleId		:= MemModIdMB;
					MDP_Read.stMDP_DynAddr.nTableId			:= 16#01;
					MDP_Read.stMDP_DynAddr.nSubIdx			:= 10;
					dwData[1]								:= 0;	
					TON_Cycle.IN							:= MDP_Read.stMDP_DynAddr.nModuleId > 0;			
					state									:= 11;
								
				11: 
					MB_Temp									:= WORD_TO_INT(dwData[1]); //Daten sichern
					
					i 										:= MIN_VOLTAGE;	
					IF Voltage_Count > 0
					THEN					
						MDP_Read.stMDP_DynAddr.nModuleId	:= MemModIdMB;
						MDP_Read.stMDP_DynAddr.nTableId		:= 16#05;
						MDP_Read.stMDP_DynAddr.nSubIdx		:= MemMBSubIdxVoltage[i];
						TON_Cycle.IN						:= MDP_Read.stMDP_DynAddr.nModuleId > 0;	
					ELSE
						dwData[1]							:= 0;	
					END_IF						
					
					state									:= 12;		
			
				12:
					MB_Voltage[i]							:= WORD_TO_INT(dwData[1]); //Daten sichern
				
					i 										:= i + 1;	
					IF i > Voltage_Count
					THEN //CPUTemp lesen 
						i									:= MIN_CPU;
						MDP_Read.stMDP_DynAddr.nModuleId	:= MemModIdCPU[i];
						MDP_Read.stMDP_DynAddr.nTableId		:= 16#01;
						MDP_Read.stMDP_DynAddr.nSubIdx		:= 3;
						TON_Cycle.IN						:= MDP_Read.stMDP_DynAddr.nModuleId > 0;		
						state								:= 13;					
					ELSE //weiter Voltage lesen
						MDP_Read.stMDP_DynAddr.nModuleId	:= MemModIdMB;
						MDP_Read.stMDP_DynAddr.nTableId		:= 16#05;
						MDP_Read.stMDP_DynAddr.nSubIdx		:= MemMBSubIdxVoltage[i];	
						TON_Cycle.IN						:= MDP_Read.stMDP_DynAddr.nModuleId > 0;		
					END_IF								
			
				13: 
					CPU_Temp[i]								:= WORD_TO_INT(dwData[1]);
					
					i 										:= i + 1;	
					IF i > CPU_Count //Start next read
					THEN //Fan auslesen 	
						IF Fan_Count > 0
						THEN
							i								:= MIN_FAN;
							
							MDP_Read.stMDP_DynAddr.nModuleId:= MemModIdFan[i];
							MDP_Read.stMDP_DynAddr.nTableId	:= 16#01;
							MDP_Read.stMDP_DynAddr.nSubIdx	:= 1;		
							TON_Cycle.IN					:= MDP_Read.stMDP_DynAddr.nModuleId > 0;			
						ELSE
							dwData[1]						:= 0;				
						END_IF
						
						state								:= 14;
						
					ELSE //CPU weiter auslesen
						MDP_Read.stMDP_DynAddr.nModuleId	:= MemModIdCPU[i];
						MDP_Read.stMDP_DynAddr.nTableId		:= 16#01;
						MDP_Read.stMDP_DynAddr.nSubIdx		:= 3;		
						TON_Cycle.IN						:= MDP_Read.stMDP_DynAddr.nModuleId > 0;						
					END_IF			
				
				14: 
					FAN_Speed[i]							:= WORD_TO_INT(dwData[1]);
					
					i 										:= i + 1;	
					IF i > Fan_Count
					THEN //CPU Usage auslesen
						(*
						i									:= MIN_CPU;
						MDP_Read.stMDP_DynAddr.nModuleId	:= MemModIdCPU[i];
						MDP_Read.stMDP_DynAddr.nTableId		:= 16#01;
						MDP_Read.stMDP_DynAddr.nSubIdx		:= 2;
						*)
						TON_Cycle.IN						:= MDP_Read.stMDP_DynAddr.nModuleId > 0;		
					//	state								:= 15;
						state								:= 90;	//final state in this section		
					
					ELSE //Fan weiter auslesen
						MDP_Read.stMDP_DynAddr.nModuleId	:= MemModIdFan[i];
						MDP_Read.stMDP_DynAddr.nTableId		:= 16#01;
						MDP_Read.stMDP_DynAddr.nSubIdx		:= 1;
						TON_Cycle.IN						:= MDP_Read.stMDP_DynAddr.nModuleId > 0;						
					END_IF				
				
				(*
				15:
					CPU_Usage[i]							:= WORD_TO_USINT(dwData[1]);
					
					i 										:= i + 1;	
					IF i > CPUCount
					THEN //Ups status auslesen 	
						IF MEmModIdUPS <> 0
						THEN
							MDP_Read.stMDP_DynAddr.nModuleId:= MEmModIdUPS;
							MDP_Read.stMDP_DynAddr.nTableId	:= 16#01;
							MDP_Read.stMDP_DynAddr.nSubIdx	:= 7;	
							TON_Cycle.IN					:= MDP_Read.stMDP_DynAddr.nModuleId > 0;
						ELSE
							dwData[1]						:= 0;								
						END_IF					
						state								:= 16;	
						
					ELSE //CPU weiter auslesen
						MDP_Read.stMDP_DynAddr.nModuleId	:= MemModIdCPU[i];
						MDP_Read.stMDP_DynAddr.nTableId		:= 16#01;
						MDP_Read.stMDP_DynAddr.nSubIdx		:= 2;		
						TON_Cycle.IN						:= MDP_Read.stMDP_DynAddr.nModuleId > 0;						
					END_IF	
			
				16:
					UPS_PowerStatus							:= WORD_TO_INT(dwData[1]);
					state									:= state * -1;	
				*)
				ELSE //90			
					Valid									:= TRUE;
					ExecutionTime	 						:= TIME() - MemTimeStartCycle;
					MemTimeStartCycle 						:= T#0MS;
					state									:= 10;	
				END_CASE
			END_IF
			TON_Cycle(PT := CycleTime);
			MDP_Read(bExecute := TON_Cycle.Q,	pDstBuf	:= ADR(dwData), cbDstBufLen := SIZEOF(dwData));
			
			IF MDP_Read.bExecute 
			THEN 
				TON_Cycle(IN := FALSE); 		
			END_IF 
			
			IF MemTimeStartCycle = T#0MS
			THEN
				MemTimeStartCycle 							:= TIME();	
			END_IF
			
		END_IF
			
	//Error State	
	99:	
		; //Wait for disable
				
	ELSE
		;
	END_CASE
ELSE //Not Enable
	state													:= 0;
	Error													:= FALSE;
	ErrorId													:= 0;
	ErrorGrp												:= eMDP_Err_NoError;
	Busy													:= FALSE;
	Valid													:= FALSE;
	MDP_Read(bExecute := FALSE);

END_IF			

(****************************************************************************************************)

END_FUNCTION_BLOCK

// POUs/IpcDiag/MDP/MDP_IpcDiag_wEvents
{attribute 'no_check'}
//General IPC diagnosis based on Beckhoff MDP - invalid values are reported via EventLogger 
//based on Tc2_MDP.lib - please see Beckhoff documentation for further information about Tc2_MDP.lib (IPC diagnostics)
//EventHandlingGrp10 instance used inside
//Info:
// 0x   	a    	nn   	x   
// 0x   	8   	03   	1   
// a 	= Area Code (e.g. 8 = Configuration Area) 
// nn 	= Modul-ID (e.g. dynamic modul id from list F020) 
// x	= Tabel id (e.g. 1 = Table 0x8nn1 - NIC Properties at area code 8) 
FUNCTION_BLOCK MDP_IpcDiag_wEvents EXTENDS MDP_IpcDiag         									
VAR_INPUT               									
	ConfirmTrig												:	BOOL := FALSE;	//Resets error with rising edge
	SourceId												:	UDINT := 100001; //EventLogger source id - Initinal value collaborates with SOURCE_ID structure 

END_VAR                 									
VAR_OUTPUT              							
	EventStatus												:	DWORD;	//state of event
END_VAR	
VAR
(* function-blocks *****************************************************************)
	Event													:	EventHandlingGrp10:= (  
																	No := [(Class := TC2_SYSTEM.TCEVENTCLASS_ALARM),
																			(Class := TC2_SYSTEM.TCEVENTCLASS_ALARM),
																			(Class := TC2_SYSTEM.TCEVENTCLASS_ALARM),
																			(Class := TC2_SYSTEM.TCEVENTCLASS_ALARM),
																			(Class := TC2_SYSTEM.TCEVENTCLASS_ALARM),
																			(Class := TC2_SYSTEM.TCEVENTCLASS_ALARM),
																			(Class := TC2_SYSTEM.TCEVENTCLASS_ALARM),
																			(Class := TC2_SYSTEM.TCEVENTCLASS_ALARM),
																			(Class := TC2_SYSTEM.TCEVENTCLASS_WARNING),
																			(Class := TC2_SYSTEM.TCEVENTCLASS_WARNING)]);
	
(* internal used variables **********************************************************)

END_VAR

(* MDP IPC diag compact						V1.1	*)
(****************************************************)

(* call base *******************************************************)
	SUPER^();

	//Leave error state by confirm trigger too
	IF State = 99 AND ConfirmTrig
	THEN
		state											:= 0;
		Error											:= FALSE;
		ErrorId											:= 0;
		ErrorGrp										:= eMDP_Err_NoError;
		Busy											:= FALSE;
		Valid											:= FALSE;
		MDP_Read(bExecute := FALSE);						
	END_IF
	
(* Meldungen *******************************************************)
	_callEvents();

(******************************************************************)

METHOD _callEvents : BOOL
VAR_INPUT
END_VAR
	IF state = 90 
		OR ConfirmTrig AND Valid
	THEN //Nur nach lesen Ende auswerten
		event.no[1].Flag 									:= FALSE ; 
		event.no[2].Flag 									:= MAX(CPU_Temp[1],CPU_Temp[2]) > MaxTempCPU; event.no[2].Text1 := INT_TO_STRING(MAX(CPU_Temp[1],CPU_Temp[2])); 
		event.no[3].Flag 									:= MB_Temp > MaxTempMB; event.no[3].Text1 := INT_TO_STRING(MB_Temp); 
	
		IF Fan_Count > 0
		THEN
			event.no[4].Flag := FALSE;
			FOR k := MIN_FAN TO MIN(Fan_Count,MAX_FAN)
			DO
				IF FAN_Speed[k] < MinSpeedFan 
					AND_THEN GETBIT32(TO_DWORD(FanMask), TO_SINT(k-1)) //Only check for active marked fans
				THEN
					event.no[4].Text1 						:= INT_TO_STRING(k); 
					event.no[4].Text2 						:= INT_TO_STRING(FAN_Speed[k]); 				
					event.no[4].Flag 						:= TRUE;
					EXIT;
				END_IF
			END_FOR		 
		ELSE
			event.no[4].Flag 								:= FALSE;
		END_IF
		
		IF Voltage_Count > 0
		THEN
			event.no[5].Flag 								:= FALSE;
			FOR k := MIN_VOLTAGE TO MIN(MAX_VOLTAGE,Voltage_Count)
			DO
				IF MB_NominalVoltage[k] <> 0
					AND(
					INT_TO_LREAL(MB_Voltage[k]) < INT_TO_LREAL(MB_NominalVoltage[k]) * VoltageFactor
					OR INT_TO_LREAL(MB_Voltage[k]) > INT_TO_LREAL(MB_NominalVoltage[k]) * (1.0 + (1.0 - VoltageFactor)))
				THEN
					event.no[5].Text1 						:= INT_TO_STRING(MB_Voltage[k]); 
					event.no[5].Text2 						:= INT_TO_STRING(MB_NominalVoltage[k]); 				
					event.no[5].Flag 						:= TRUE;
					EXIT;
				END_IF
			END_FOR		 
		ELSE
			event.no[5].Flag 								:= FALSE;
		END_IF
	
		event.no[6].Flag 									:= FALSE;
		event.no[7].Flag 									:= FALSE; 
		event.no[8].Flag 									:= FALSE; 
		event.no[9].Flag 									:= MAX(CPU_Temp[1],CPU_Temp[2]) > MaxTempCPU - TempWarningThreshold ; event.no[9].Text1 := INT_TO_STRING(MAX(CPU_Temp[1],CPU_Temp[2])); 
		event.no[10].Flag 									:= MB_Temp > MaxTempMB - TempWarningThreshold; event.no[10].Text1 := INT_TO_STRING(MB_Temp); 
	END_IF
	
	Event(
		ConfirmTrig	:= ConfirmTrig,
		SourceId	:= SourceId,
		no			:= ,
		Disable		:= NOT Enable,
		AutoConfirm := ,
		MIN_EVENT	=> ,
		MAX_EVENT	=> ,
		Status		=> EventStatus);
END_METHOD

END_FUNCTION_BLOCK

// POUs/IpcDiag/UPSStatus
{attribute 'no_check'}
//General UPS function block to make use of differenty types of utility power supplies 
//Requiered libs : Tc2_SUPS, Tc2_IoFunctions
FUNCTION_BLOCK UPSStatus
VAR_OUTPUT CONSTANT
	MODE_SUPS_CB3011										:	INT := 0; //SUPS for CB3011 Motherboard
	MODE_SUPS_CX50X0										:	INT := 1; //SUPS for CX50X0
	MODE_SUPS_CX51X0										:	INT := 2; //SUPS for CX51X0
	MODE_SUPS_CX9020										:	INT := 3; //SUPS for CX9020
	MODE_SUPS_BAPI											:	INT := 4; //SUPS for BAPI
	MODE_UPS_BA												:	INT := 5; //BA UPS Controller CP903x-Card (PCI/ISA) | Beckhoff P24Vxxxx USV | With Beckhoff Industrial PC's delivered APC UPS models supporting smart protocol and configured with Windows UPS Service
	MODE_UPS_EXTERN_OK										:	INT := 6; //External UPS controller connected via one Digital Input -> TRUE=PowerOK
	MODE_UPS_EXTERN_FAIL									:	INT := 7; //External UPS controller connected via one Digital Input -> TRUE=PowerFAIL
END_VAR                     								
VAR_INPUT                   													
	Enable													: 	BOOL := FALSE;		// FB will be processed as long as enable is TRUE 
	NetId													: 	T_AmsNetId 	:= '';	// AmsNet id
	Port													: 	T_AmsPort 	:= 851; // TC3 PLC RT1 = 851.... , 0 = Windows UPS service 
	Timeout													: 	TIME := DEFAULT_ADS_TIMEOUT; // Ads timeout / PowerOK/Fault delay at mode = MODE_UPS_EXTERN
	Mode													: 	INT(MODE_SUPS_CB3011..MODE_UPS_EXTERN_FAIL) := MODE_UPS_BA; // Select used UPS type
	UpsMode													: 	E_S_UPS_Mode := eSUPS_WrPersistData_Shutdown; // Used by FB_S_UPS instances and adaped for modes <> MODE_SUPS  
END_VAR
VAR_OUTPUT
	BatteryReplace											:	BOOL;
	PowerFailDetect											:	BOOL; 	//TRUE when power fail is detected 
	Status													:	E_S_UPS_State := eSUPS_PowerOK; //Reports the status of utility-supplied power into the UPS. 
	Error													:	BOOL;		//Rising edge of Error informs that an error occurred during the execution of the Function Block  	
{attribute 'displaymode':='hex'}
	ErrorID													:	UDINT; 	//Error identification 
END_VAR      
VAR              
//local *****************************************************************
	State													: 	INT := 0;
	DigInput										AT %I*	: 	BOOL; //Hardware signal for OK/NOK depending on selected UpsMode
	
//Trigger ***************************************************************

//Timer ****************************************************************
	TonPowerOff												: 	TON;	
//Instances **********************************************************  
	UPSPowerStatus											: 	FB_GetUpsStatus;
	SUPSPowerStatus_CB3011									: 	FB_S_UPS_CB3011 		:= (ePersistentMode := SPDM_2PASS);
	SUPSPowerStatus_CX50X0									: 	FB_S_UPS 				:= (iUPSPort := 16#4A8 ,ePersistentMode := SPDM_2PASS);	
	SUPSPowerStatus_CX51x0									: 	FB_S_UPS_CX51x0 		:= (iUPSPort := 16#588 ,ePersistentMode := SPDM_2PASS);
	SUPSPowerStatus_CX9020									: 	FB_S_UPS_CX9020_U900 	:= (ePersistentMode := SPDM_2PASS);
	SUPSPowerStatus_BAPI									: 	FB_S_UPS_BAPI			:= (ePersistentMode := SPDM_2PASS);
	ShutDown												: 	NT_Shutdown;
	WritePersistentData										: 	FB_WritePersistentData := (Mode := SPDM_2PASS);	
	TcStop													: 	TC_Stop;
//Dummy *****************************************************************)       								

END_VAR

	(* UPS Wrapper										*)
	(****************************************************)

(* Sequence *************************************************************************)
IF Enable THEN
	CASE state OF	
	0:
		CASE MODE OF
		MODE_SUPS_CB3011:
			SUPSPowerStatus_CB3011(
				sNetID				:= NetId,
				iPLCPort			:= Port,
				tTimeout			:= ,
				eUpsMode			:= UpsMode,
				ePersistentMode		:= ,
				tRecoverTime		:= ,
				bPowerFailDetect	=> PowerFailDetect,
				eState				=> Status);		
		
		MODE_SUPS_CX50X0:
			SUPSPowerStatus_CX50X0(
				sNetID				:= NetId,
				iPLCPort			:= Port,
				iUPSPort			:= ,
				tTimeout			:= ,
				eUpsMode			:= UpsMode,
				ePersistentMode		:= ,
				tRecoverTime		:= ,
				bPowerFailDetect	=> PowerFailDetect,
				eState				=> Status);		
			
		MODE_SUPS_CX51X0:
			SUPSPowerStatus_CX51x0(
				sNetID				:= NetId,
				iPLCPort			:= Port,
				iUPSPort			:= ,
				tTimeout			:= ,
				eUpsMode			:= UpsMode,
				ePersistentMode		:= ,
				tRecoverTime		:= ,
				bPowerFailDetect	=> PowerFailDetect,
				eState				=> Status);		
			
		MODE_SUPS_CX9020:
			SUPSPowerStatus_CX9020(
				sNetID				:= NetId,
				iPLCPort			:= Port,
				tTimeout			:= ,
				eUpsMode			:= UpsMode,
				ePersistentMode		:= ,
				tRecoverTime		:= ,
				bPowerFailDetect	=> PowerFailDetect,
				eState				=> Status);		
				
		MODE_SUPS_BAPI:
			SUPSPowerStatus_BAPI(
				sNetID				:= NetId,
				iPLCPort			:= Port,
				tTimeout			:= ,
				eUpsMode			:= UpsMode,
				ePersistentMode		:= ,
				tRecoverTime		:= ,
				bPowerFailDetect	=> PowerFailDetect,
				eState				=> Status);				

		MODE_UPS_EXTERN_OK,
		MODE_UPS_EXTERN_FAIL:
			TonPowerOff(
				IN					:= SEL(MODE = MODE_UPS_EXTERN_OK, DigInput, NOT DigInput), 
				PT					:= Timeout, 
				Q 					=> PowerFailDetect);
			Status											:= SEL(TonPowerOff.IN, eSUPS_PowerOK, eSUPS_WaitForRecover);
			IF TonPowerOff.Q                                
			THEN				                            
				Status										:= eSUPS_PowerFailure;
				state										:= 900;
			END_IF 
			
		MODE_UPS_BA:		
			UPSPowerStatus(
				sNetId				:= NetId, 
				nPort				:= 0, 
				bEnable				:= TRUE, 
				bValid				=> , 
				bError				=> Error, 
				nErrId				=> ErrorID);
			BatteryReplace									:= UPSPowerStatus.stStatus.eBatteryStatus = E_BatteryStatus.BatteryReplace AND UPSPowerStatus.bValid;
			CASE UPSPowerStatus.stStatus.ePowerStatus OF 
			PowerUnknownStatus: 			// The status of power is unknown
				PowerFailDetect								:= FALSE;
				Status										:= eSUPS_PowerOK;	
 			PowerOnLine: 		 		  	// Power is OK
				PowerFailDetect								:= FALSE;
				Status										:= eSUPS_PowerOK;
   			PowerOnBattery:					// A power failure has occurred
				PowerFailDetect								:= UPSPowerStatus.bValid;
				Status										:= eSUPS_PowerFailure;
				state										:= 900;
			END_CASE
	
		ELSE
			state											:= 0;
			Error											:= TRUE;
			ErrorID											:= 1798;	
			PowerFailDetect									:= FALSE;		
			Status											:= eSUPS_PowerFailure;		
		END_CASE
		
	//Shutdown OS and stop TC ************************************************************)
	900: 
		ShutDown(START := FALSE); TcStop(Stop := FALSE); WritePersistentData(Start := FALSE);
		CASE UpsMode OF
		eSUPS_WrPersistData_NoShutdown:
			WritePersistentData(Start := TRUE, Port := Port);		
			status											:= eSUPS_WritePersistentData;
		eSUPS_ImmediateShutdown:
			ShutDown(START := TRUE, TMOUT := T#3S); 
			status											:= eSUPS_QuickShutdown;			
		ELSE //eSUPS_WrPersistData_Shutdown
			ShutDown(START := TRUE, TMOUT := T#3S);
			status											:= eSUPS_WritePersistentData;
		END_CASE
		state												:= state + 1;	
											
	901:// Wait for shutdown started     
		shutDown();  WritePersistentData();  																		
		IF ShutDown.BUSY OR ShutDown.ERR OR NOT WritePersistentData.BUSY         				
		THEN                   
			Error											:= WritePersistentData.ERR OR ShutDown.ERR;
			ErrorId											:= SEL(WritePersistentData.ERR, ShutDown.ERRID , WritePersistentData.ERRID);
			IF UpsMode = eSUPS_ImmediateShutdown
			THEN
				status										:= eSUPS_WaitForPowerOFF;
			ELSIF UpsMode = eSUPS_WrPersistData_NoShutdown
			THEN
				status										:= eSUPS_WaitForRecover;
				state										:= 0;
			ELSE //Stop TC and write persistent data
				state										:= state + 1;
			END_IF		
		END_IF                          				
													
	902:(*Tc Stop*)                       	
		TcStop(STOP := TRUE);
		IF NOT TcStop.BUSY
		THEN
			Error											:= Error OR TcStop.ERR;
			ErrorId											:= SEL(TcStop.ERR, ErrorId, TcStop.ERRID);
			status											:= eSUPS_WaitForPowerOFF;
		END_IF
			
	END_CASE

ELSE
	Status													:= eSUPS_PowerOK;
	state													:= 0;
	Error													:= FALSE;
	ErrorID													:= 0;	
	PowerFailDetect											:= FALSE;
END_IF

(********************************************************************)

END_FUNCTION_BLOCK

// POUs/Logging/adsLogError
{attribute 'no_check' := ''}
//Writes a string as a error message into the TwinCAT AMS Logger and Windows Event Log with an possible argument
//Please see Beckhoff information system "ADSLOGxxxx" for detailed information.
//Intention of this function is to use the handy ADSLOGxxxx with a predefined msgCtrlMask of "ADSLOG_MSGTYPE_STRING OR ADSLOG_MSGTYPE_HINT OR ADSLOG_MSGTYPE_LOG"
FUNCTION adsLogError : DINT //Write error message into ADS log windows - Return value will be error code or 0 if OK
VAR_INPUT               											
	MsgFmtStr												:	T_MaxString; //Message text with %s as placeholder for StrArg
(*	dintArg													:	DINT; //DINT argument for message - to be replaced by %d *) 
	StrArg													:	T_MaxString; //String argument for message - to be replaced by %s
(*	realArg													:	LREAL; //LREAL argument for message - to be replaced by %f *) 
END_VAR
VAR
	msgCtrlMask												:	DWORD; (* 	ADSLOG_MSGTYPE_HINT Meldungstyp ist Hinweis.
																				ADSLOG_MSGTYPE_WARN Meldungstyp ist Warnung.  
																				ADSLOG_MSGTYPE_ERROR Meldungstyp ist Fehler.  
																				ADSLOG_MSGTYPE_LOG Meldung wird in das Logbuch geschrieben.  
																				ADSLOG_MSGTYPE_MSGBOX Meldung wird in einer Messagebox ausgegeben.  
																				ADSLOG_MSGTYPE_RESOURCE Meldung wird aus einer Ressource-Datei geholt. (wird momentan nicht  unterstützt)  
																				ADSLOG_MSGTYPE_STRING 	Meldung ist direkt angegebener String (default).  *)	
END_VAR

(* create fixed message ctrl mask **********************************)
	msgCtrlMask												:= ADSLOG_MSGTYPE_STRING OR ADSLOG_MSGTYPE_ERROR OR ADSLOG_MSGTYPE_LOG;

(* write string which includes a floating-number ******************)
(*	AdsLogError 											:= ADSLOGLREAL(msgCtrlMask, msgFmtStr, realArg); *)
	
(* write string which includes a DINT-number *******************)
(*	AdsLogError 											:= ADSLOGDINT(msgCtrlMask, msgFmtStr, dintArg); *)

(* write string which includes an other string e.g. 'hallo: %s what's up' ***************)
	adsLogError 											:= ADSLOGSTR(msgCtrlMask, msgFmtStr,strArg); 

(*****************************************************)

END_FUNCTION

// POUs/Logging/I_LogbookSubscriber
INTERFACE I_LogbookSubscriber Extends __System.IQueryInterface

METHOD addNewMessage : BOOL
VAR_IN_OUT
	data										:	LogbookData;
END_VAR
END_METHOD

{attribute 'monitoring' := 'call'}
PROPERTY PUBLIC isBusy : BOOL
GET
END_GET
END_PROPERTY

END_INTERFACE

// POUs/Logging/LogbookPuplisher
{attribute 'no_check' := ''}
//The LogbookPuplisher checks the used logbook for new entrys and those to his subscribers
FUNCTION_BLOCK LogbookPuplisher
VAR CONSTANT 
	MIN_SUBSCRIBERS											:	INT := 1;
	MAX_SUBSCRIBERS											:	INT := PARAM.LOGBOOK_PUPLISHER_MAX_SUB;	
END_VAR                     								
VAR_INPUT                   								
	Enable													: 	BOOL; //Enable logbook server
	ipLogbookSubscribers									: 	ARRAY[MIN_SUBSCRIBERS..MAX_SUBSCRIBERS] OF I_LogbookSubscriber;
END_VAR                     								
VAR_IN_OUT                  								
	SystemTime												: 	TIMESTRUCT; //System time - written to the logbook timestamp if it is not updated externally
	Book													: 	Logbook; //Logbook instance
END_VAR                     								
VAR_OUTPUT                
	LastEntry												: 	LogbookData;	  								
	Busy													: 	BOOL; //New message occured
END_VAR                     								
VAR            
//local ************************************************************************************

//trigger *********************************************************************************

//timer ***********************************************************************************

//instances ***********************************************************************************             								

//Dummys ****************************************************************************************
	i,j														: INT;
	k														: UINT;
END_VAR

	(* Logbook server								*)
	(************************************************)

(* Check new Entrys ***************************************************)
Busy														:= FALSE;
Book.Timestamp												:= SystemTime; //Update Logbook timestamp
IF Enable 
THEN
	FOR i := Book.MIN_DATA TO Book.CntAddedMessages
	DO //Add new messages to subrscruber as long as they are not busy or until all new messages are read
		IF NOT subscriberBusy AND_THEN Book.getOldestMsg(LastEntry)
		THEN
			Busy											:= TRUE;
			IF LastEntry.Timestamp.wDay = 0
			THEN //Add timestamp to Entry if empty
				LastEntry.Timestamp							:= SystemTime;
			END_IF
			
			FOR j := MIN_SUBSCRIBERS TO MAX_SUBSCRIBERS
			DO
				IF ipLogbookSubscribers[j] <> 0
				THEN
					ipLogbookSubscribers[j].addNewMessage(LastEntry);
				ELSE
					EXIT;
				END_IF
			END_FOR
		ELSE
			EXIT;
		END_IF
	END_FOR
END_IF
(**************************************************************************)

PROPERTY PRIVATE subscriberBusy : BOOL
GET
VAR
	 i : INT;
END_VAR
SubscriberBusy									:= FALSE;
FOR i := MIN_SUBSCRIBERS TO MAX_SUBSCRIBERS
DO
	IF ipLogbookSubscribers[i] <> 0
	THEN
		IF ipLogbookSubscribers[i].IsBusy
		THEN
			SubscriberBusy						:= TRUE;
			EXIT;
		END_IF
	ELSE
		EXIT;
	END_IF
END_FOR
END_GET
END_PROPERTY

END_FUNCTION_BLOCK

// POUs/Logging/LogbookSubEventLog
//{attribute 'no_check' := ''}
//The LogbookSubEventLog sends log entries from the LogbookPuplisher to the EventLogger
//Include instances of EventHandling and needs "LogbookServer" as parameter  
FUNCTION_BLOCK LogbookSubEventLog IMPLEMENTS I_LogbookSubscriber
VAR CONSTANT 
	MIN_EVENT												: UINT := 1;
	MAX_EVENT												: UINT := PARAM.LOGBOOK_SUB_MAX_EVENT_HANDLING; //see library parameter to customize parameter	
END_VAR                     								
VAR_INPUT                   								
	Enable													: BOOL; //Enable
	ConfirmEvents											: BOOL; //Quitting for corresponding event classes / set to TRUE for an auto quitting of messages which are gone
	SourceID												: UDINT := 0; //TcEventLogger source id
	PT_ShowEventLog											: TIME := TIME#5S; //Display time for logbook entrys that dont need to be reseted 
END_VAR                     								
VAR_IN_OUT                  								
END_VAR                     								
VAR_OUTPUT          
	Busy													: BOOL; //Write msg to file or display via tcEventLogger is active       								
	Error													: BOOL;
{attribute 'displaymode':='hex'}
	ErrorId													: UDINT; //Ads error 16#708 busy if all events are occuopied	
END_VAR                     								
VAR            
//local ************************************************************************************
	State													: INT := 0;
	NextEvent												: UINT := MIN_EVENT;
	MsgString												: ARRAY[MIN_EVENT..MAX_EVENT] OF STRING(PARAM.LOGBOOK_MAX_MSG_STRING_LENGHT);

	CntAllEventsOccpied										:	INT;
	
//trigger *********************************************************************************


//timer ***********************************************************************************
	tofShowMsg												: ARRAY[MIN_EVENT..MAX_EVENT] OF TOF;

//instances ***********************************************************************************             								
	EventNo													: ARRAY[MIN_EVENT..MAX_EVENT] OF EventHandling;	

//Dummys ****************************************************************************************
	i,j														: UINT;
	k														: UINT;
END_VAR

	(* Logbook subscriber - logbook entries send to Eventlogger			*)
	(********************************************************************)

(* show messages via Eventlogger ***************************************)
	NextEvent												:= 0;
	FOR i := MIN_EVENT TO MAX_EVENT 
	DO
		tofShowMsg[i](IN := FALSE, Q => EventNo[i].Flag);
		IF EventNo[i].State <> TCEVENTSTATE_INVALID OR EventNo[i].Flag 
		THEN
			EventNo[i](ConfirmTrig	:= ConfirmEvents OR NOT tofShowMsg[i].q AND EventNo[i].State <> TCEVENTSTATE_INVALID, SourceId := SourceId);
		ELSE
			NextEvent										:= i;
		END_IF
	END_FOR

(* Status ****************************************************************)
	Busy													:= NextEvent = 0; //No more event free to trigger

(* Ack ErrorIds **********************************************************)
	IF ConfirmEvents 
	THEN
		CntAllEventsOccpied									:= 0;
		Error												:= FALSE;
		ErrorId												:= 0;
	END_IF
                      							
(*************************************************************************)

METHOD PUBLIC FINAL addNewMessage : BOOL //Return value = TRUE if execution successful finished
VAR_IN_OUT
	data													:	LogbookData;
END_VAR
	IF NextEvent >= MIN_EVENT and NextEvent <= MAX_EVENT
	THEN
		MsgString[NextEvent]								:= Data.Msg;
		EventNo[NextEvent].Class.0							:= Data.Options.8; 
		EventNo[NextEvent].Class.1							:= Data.Options.9; 
		EventNo[NextEvent].Class.2							:= Data.Options.10; 
		EventNo[NextEvent].Class.3							:= Data.Options.11; 
		
		tofShowMsg[NextEvent](IN := Enable, PT := PT_ShowEventLog);
		NextEvent											:= 0;
		addNewMessage										:= TRUE;
	ELSE
		addNewMessage										:= FALSE;
		CntAllEventsOccpied									:= CntAllEventsOccpied + 1;
		ErrorId												:= 16#0708; //Busy
	END_IF
END_METHOD

METHOD FB_init : BOOL
VAR_INPUT
	bInitRetains : BOOL; // if TRUE, the retain variables are initialized (warm start / cold start)
	bInCopyCode : BOOL;  // if TRUE, the instance afterwards gets moved into the copy code (online change)
END_VAR
	FOR i := MIN_EVENT TO MAX_EVENT 
	DO
		EventNo[i].MsgId									:= TO_UINT(i);
		EventNo[i].pText3									:= ADR(MsgString[i]);
	END_FOR
	
	Fb_init 												:= TRue;
END_METHOD

{attribute 'monitoring' := 'call'}
PROPERTY PUBLIC FINAL isBusy : BOOL
GET
IsBusy											:= NextEvent = 0;
END_GET
END_PROPERTY

END_FUNCTION_BLOCK

// POUs/Logging/LogbookSubSendMail
{attribute 'no_check' := ''}
//The LogbookSubSendMail sends log entries via email which are handed over by the Logbook Puplisher 
{attribute 'enable_dynamic_creation'}
FUNCTION_BLOCK LogbookSubSendMail IMPLEMENTS I_LogbookSubscriber
VAR CONSTANT
	MAX_BUFFER_LEVEL										:	INT := 85; //If buffer fill level reaches 85% Fb will appear as "busy2 to the LogBookPuplisher 
END_VAR
VAR_OUTPUT CONSTANT 
	STRING_LINE_END_SIGN									: STRING(6) := '$r$n'; //$r $n

{attribute 'displaymode':='binary'}
	OPTION_ADD_TIMESTAMP_TO_MSG								: BYTE := 2#0000_0001; 	
{attribute 'displaymode':='binary'}
	OPTION_SEND_STORED_MSG_WITH_DISABLE						: BYTE := 2#0010_0000; //Send stored messages if FB gets disabled to clear buffer 	
{attribute 'displaymode':='binary'}
	OPTION_ENABLE_BUFFER_ERROR								: BYTE := 2#0100_0000; //The FB changes to error state if the buffer was not emptied in time 
END_VAR                     								
VAR_INPUT                   								
	Enable													: BOOL; //Enable write log entries to file
	ResetTrig												: BOOL; //Reset internal error
{attribute 'displaymode':='binary'}
	Options													: BYTE := 2#0000_0000; // Bit 0 = Add msg timestamnp to entry string 	 
	SendByNoOfMsg											: INT := PARAM.LOGBOOK_MAX_DATA; //Collected number of messages until a mail will be send
	PT_SendByTime											: TIME := T#60M; //Delay until a mail will be send if a message occured
	LogPriorityLevel										:	UINT := 0; 		//Correlate to EventClass prioritys - see Para.EVENT_HANDLING_CONFIG prioritys
	
//Smtp parameter
	SmtpServer												: T_AmsNetID;   // Smtp Server addres ( IP or Name)                  
	Username												: T_MaxString;  // Smtp Username 
	Password												: T_MaxString;  // Smtp Password                 
	Encryption												: UDINT;        // 0=NONE, 1=STARTTLS, 2=SSL                 
	FromUser												: T_MaxString;  // Sender string
	ToNames													: T_MaxString;  // To recipient string                   
	CcNames													: T_MaxString;  // Cc recipient string           
	Subject													: T_MaxString;  // Email subject            
END_VAR                     								                 								
VAR_OUTPUT       
	CntNoOfStoredMsgs										: INT;
	TimeSendMsgs											: TIME; //Elapsed time to send messages
	Busy													: BOOL; //Write msg to file active   
	Error													: BOOL;        		
{attribute 'displaymode':='hex'}						
	ErrorId													: UDINT; 
END_VAR                     								
VAR            
//local ************************************************************************************
	State													: INT := 0;
	LastMessageData											: LogbookData;	
	LastEventClass											:	E_TcEventClass := TC2_SYSTEM.TCEVENTCLASS_NONE;
	MsgString												: T_MAxString;
	StartTimeSendMsgs										:	TIME; 
				
//trigger *********************************************************************************
	
//timer ***********************************************************************************
	tonSend													:	ton;

//instances ***********************************************************************************             								
	DblBuffer												: DoubleBuffer;    

	Smtp													: FB_SmtpV3 := (
																	sNetId         	:= '',
																	sSmtpServer     := '',  (* Smtp Server addres ( IP or Name) *)
																	sUsername       := '',  (* Smtp Username *)
																	sPassword       := '',  (* Smtp Password *)
																	nEncryption     := 0,   (* 0=NONE, 1=STARTTLS, 2=SSL *)
																	sFrom           := '',	(* Sender string *)
																	sTo             := '',  (* To recipient string *)
																	sCc             := '',  (* Cc recipient string *)
																	sBcc            := '', (* Bcc recipient string *)
																	sSubject        := '', (* Subject string *)
																	tTimeout        := T#20S);


//Dummys ****************************************************************************************
	i,j														: INT;
END_VAR

	(* Logbook subscriber send mail 						*)
	(********************************************************)

(* Sequence started by method "NewMessage" ***************************************************)
	CASE State OF
	0:	
		IF Error
		THEN
			IF ResetTrig OR NOT Enable
			THEN
				Error										:= FALSE;
				ErrorId										:= 0;
				Smtp(bExecute := FALSE);
			END_IF
		ELSIF Enable
		THEN 
			DblBUffer.SizeOfMemory							:= TO_UDINT(SendByNoOfMsg) * SIZEOF(MsgString) * 2;
			
			tonSend(IN := PT_SendByTime > T#0MS AND CntNoOfStoredMsgs > 0, PT := PT_SendByTime);
			
			IF NOT DblBuffer.ReadyToRead 
				AND(tonSend.Q OR CntNoOfStoredMsgs > SendByNoOfMsg)
			THEN 
				DblBuffer.setReadyToRead(TRUE);
			END_IF
			
			IF DblBuffer.ReadyToRead 			
			THEN
				tonSend(IN := FALSE);
				CntNoOfStoredMsgs							:= 0;
				StartTimeSendMsgs							:= TIME();
				
				Smtp(
					sNetId		:= , 
					sSmtpServer	:= SmtpServer, 
					sUsername	:= Username, 
					sPassword	:= Password, 
					nEncryption	:= Encryption, 
					sFrom		:= FromUser, 
					sTo			:= ToNames, 
					sCc			:= CcNames, 
					sBcc		:= , 
					sSubject	:= Subject, 
					pMessage	:= DblBuffer.pDataToRead, 
					cbMessage	:= DblBuffer.SizeOfDataToRead, 
					bExecute	:= TRUE, 
					tTimeout	:= , 
					bBusy		=> , 
					bError		=> , 
					nErrId		=> );
													
				state										:= 1;
			END_IF
		ELSE //not enabled
			IF NOT DblBuffer.Empty AND Options.5
			THEN //Write rest of buffer
				IF NOT DblBuffer.ReadyToRead THEN DblBuffer.setReadyToRead(TRUE); END_IF 
				Smtp(
					sNetId		:= , 
					sSmtpServer	:= SmtpServer, 
					sUsername	:= Username, 
					sPassword	:= Password, 
					nEncryption	:= Encryption, 
					sFrom		:= FromUser, 
					sTo			:= ToNames, 
					sCc			:= CcNames, 
					sBcc		:= , 
					sSubject	:= Subject, 
					pMessage	:= DblBuffer.pDataToRead, 
					cbMessage	:= DblBuffer.SizeOfDataToRead, 
					bExecute	:= TRUE, 
					tTimeout	:= , 
					bBusy		=> , 
					bError		=> , 
					nErrId		=> );
				CntNoOfStoredMsgs							:= 0;
				StartTimeSendMsgs							:= TIME();
				State										:= 1;
			END_IF
		END_IF
				
	1:
		Smtp(bExecute	:= TRUE, pMessage := DblBuffer.pDataToRead,  cbMessage := DblBuffer.SizeOfDataToRead);
		IF NOT Smtp.bBusy
		THEN
			IF Smtp.bError
			THEN
				Error										:= TRUE;
				ErrorId										:= Smtp.nErrId;
				State										:= 0;
			ELSE				
				State										:= 0;
			END_IF 
			DblBuffer.setReadyToRead(FALSE);	
			TimeSendMsgs									:= TIME() - StartTimeSendMsgs;
			Smtp(bExecute	:= FALSE);
		END_IF 
	ELSE
		;
	END_CASE

(* Ack ErrorIds **********************************************************)
	Busy 													:= State <> 0;
(**************************************************************************)

METHOD PUBLIC FINAL addNewMessage : BOOL //Return value = TRUE if execution successful finished
VAR_IN_OUT
	data													:	LogbookData;
END_VAR
	
	IF Enable AND NOT Error
	THEN	
		LastMessageData										:= Data;
		LastEventClass.0									:= LastMessageData.Options.8;
		LastEventClass.1									:= LastMessageData.Options.9;
		LastEventClass.2									:= LastMessageData.Options.10;
		LastEventClass.3									:= LastMessageData.Options.11;
			
		//Copy messages to memory	
		IF LogPriorityLevel = 0 OR_ELSE GetEventClassPriority(LastEventClass) > LogPriorityLevel
		THEN	
			MEMSET(ADR(MsgString),0,SIZEOF(MsgString));										
			IF 1 = (Options AND OPTION_ADD_TIMESTAMP_TO_MSG) 					
			THEN
				MsgString									:=	SYSTEMTIME_TO_STRING(LastMessageData.Timestamp);
				MsgString									:=	MID(MsgString, 12 , 12);
				MsgString 									:=	CONCAT(MsgString, ' | ');
			END_IF                          	
			MsgString 										:= 	CONCAT(MsgString, LastMessageData.Msg);
			MsgString 										:= 	CONCAT(MsgString, STRING_LINE_END_SIGN);

			//Add msg to memory
			CntNoOfStoredMsgs								:= CntNoOfStoredMsgs + 1;
			
			IF DblBuffer.addString(MsgString) <> S_OK
				AND Options.6
			THEN
				Error										:= TRUE;
				ErrorId										:= HRESULT_TO_ADSERROR(DblBuffer.hr);	
			END_IF	
		END_IF
	
		addNewMessage										:= NOT Error;
	ELSE
		addNewMessage										:= FALSE;
	END_IF
END_METHOD

{attribute 'monitoring' := 'call'}
PROPERTY PUBLIC FINAL isBusy : BOOL
GET
isBusy											:= DblBuffer.Full and Enable and not Error and DblBuffer.fillLevel >= MAX_BUFFER_LEVEL;
END_GET
END_PROPERTY

PROPERTY PUBLIC optAddTimeToMsg : BOOL
GET
optAddTimeToMsg := Options.0;
END_GET
SET
Options.0 := optAddTimeToMsg;
END_SET
END_PROPERTY

PROPERTY PUBLIC optEnableBufferError : BOOL
GET
optEnableBufferError := Options.6;
END_GET
SET
OPtions.6				:= optEnableBufferError;
END_SET
END_PROPERTY

PROPERTY PUBLIC optSendMsgIfDisabled : BOOL
GET
optSendMsgIfDisabled := Options.5;
END_GET
SET
Options.5 := optSendMsgIfDisabled;
END_SET
END_PROPERTY

END_FUNCTION_BLOCK

// POUs/Logging/LogbookSubSysLog
{attribute 'no_check' := ''}
//Sends Logbook entries handover by a LogbookPuplisher as SysLog messages to a SysLog Server 
//See wikipedia for more further inforamation about Syslog  
//based on TF6310 Tcp/Ip server 
FUNCTION_BLOCK LogbookSubSysLog IMPLEMENTS I_LogbookSubscriber
VAR CONSTANT
	MAX_BUFFER_LEVEL										:	INT := 85; //If buffer fill level reaches 85% Fb will appear as "busy2 to the LogBookPuplisher 
END_VAR

VAR CONSTANT 		
	MAX_SEND_STRING_SIZE									:	INT := 1024;
END_VAR
VAR_OUTPUT CONSTANT
{attribute 'displaymode':='binary'}
	OPTION_SYSLOG_WITH_FACILITY_SEVERITY_CODE				:	BYTE := 2#0000_0001;
{attribute 'displaymode':='binary'}
	OPTION_SYSLOG_WITH_RFC_HEADER							:	BYTE := 2#0000_0010;
{attribute 'displaymode':='binary'}
	OPTION_SYSLOG_WITH_CR									:	BYTE := 2#0000_0100; 
	{attribute 'displaymode':='binary'}
	OPTION_SYSLOG_WITH_LF									:	BYTE := 2#0000_1000; 
{attribute 'displaymode':='binary'}
//	OPTION_SYSLOG_WITH_TCP_MODE								:	BYTE := 2#0001_0000;
{attribute 'displaymode':='binary'}
	OPTION_SEND_STORED_MSG_WITH_DISABLE						: 	BYTE := 2#0010_0000; //Send stored messages if FB gets disabled to clear buffer
{attribute 'displaymode':='binary'}
	OPTION_ENABLE_BUFFER_ERROR								: 	BYTE := 2#0100_0000; //The FB changes to error state if the buffer was not emptied in time 	
{attribute 'displaymode':='binary'}
	OPTION_ENABLE_DEBUG										:	BYTE := 2#1000_0000; //Creates ADS log entries for conection events and errors
END_VAR
VAR_INPUT
	Enable													: 	BOOL;	//Enables sending new messages
	ResetTrig												:	BOOL;	//Ack error message
{attribute 'displaymode':='binary'}
	Options													:	BYTE := OPTION_SYSLOG_WITH_FACILITY_SEVERITY_CODE ; //option constants are alreay predefined, so they can accordingly be passed symbolically to the block
	SizeOfBuffer											:	UDINT := 2560; //Size of memory allocated from ads router memory pool by DoubleBuffer instance
	LocalHost	 											: 	T_IPv4Addr;  	//Local (client) address. String containing an (Ipv4) Internet Protocol dotted address. 
	LocalPort												:	UDINT := 515;	//Local (client) Internet Protocol (IP) port. (TCP Port = 1468) *)	
	RemoteHost	 											: 	T_IPv4Addr;  	//Remote (server) address. String containing an (Ipv4) Internet Protocol dotted address. 
	RemotePort												:	UDINT := 514;	//Remote (server) Internet Protocol (IP) port. (TCP Port = 1468) 
	Facility												:	BYTE := 16; 	//Default local 16
	Severity 												:	BYTE := 7; 		//0=Emergency/1=Alert/2=Critical/3=Error/4=Warning/5=Notice/6=Informational/7=Debug
	Tag														:	STRING(32) := ''; //Process name or local host by default
	LogPriorityLevel										:	UINT := 0; 		//Correlate to EventClass prioritys - see Para.EVENT_HANDLING_CONFIG prioritys
END_VAR                 				
VAR_OUTPUT              				        			
	Online													:	BOOL;		//TRUE if coonection is sucessful etablished
	hSocket													: 	T_HSOCKET ; //UDP Socket handle
	CntNoOfStoredMsgs										:	INT;
	TimeSendMsgs											:	TIME;
	Busy													: 	BOOL;  //Sending busy
	Error													: 	BOOL;	//Error occured
{attribute 'displaymode':='hex'}
	ErrorId													:	UDINT;	//See Beckhoff TF6310/ADS documentation for more information regarding error code
	ErrorFnc												:	STRING(20); //Error source 
	WinsockErrorId											:	E_WinsockError; //Winsocket error enum - see TF6310 documentation for further information
END_VAR
VAR
(* Memory ************************************************************)
	State													: 	INT := 0;
	StartTimeSendMsgs										:	TIME;
	SendErrorCnt											:	UINT;
	HeaderString											:	STRING;
	SendString												:	STRING(MAX_SEND_STRING_SIZE);
	SendStringLen											:	INT;
	_Severity												:	BYTE;
	LastMessageData											: 	LogbookData;
	LastEventClass											:	E_TcEventClass := TC2_SYSTEM.TCEVENTCLASS_NONE;
	
(* Trigger *****************************************************************)

(* Timer ******************************************************************)

(* Blocks ***************************************************************)
	DblBuffer												:	DoubleBuffer;
	SocketClose												:	FB_SocketClose := (tTimeout := DEFAULT_ADS_TIMEOUT);
	SocketUdpCreate 										:	FB_SocketUdpCreate := (tTimeout := DEFAULT_ADS_TIMEOUT);
	SocketUdpSend											:	FB_SocketUdpSendTo := (tTimeout := T#10S);

(* Dummys *******************************************************************)
	i,j														:	INT;
END_VAR
(* 
Facality Description:
00 Kernel message
01 user-level messages
02 mail system
03 system daemons
04 security/authorization messages
05 messages generated internally by syslogd
06 line printer subsystem
07 network news subsystem
08 UUCP subsystem
09 clock daemon
10 security/authorization messages
11 FTP daemon
12 NTP subsystem
13 log audit
14 log alert
15 clock daemon
16 local10
17 local11
18 local12
19 local13
20 local14
21 local15
22 local16
23 local17

Severity Description:
0 Emergency
1 Alert
2 Critical
3 Error
4 Warning
5 Notice
6 Informational
7 Debug
*)

(* Logbook subscriber to send sys log messages via UDP 				*)
(********************************************************************)

(* Server connection ************************************************)
	CASE state OF
	0:
		IF Error
		THEN
			IF NOT Enable OR ResetTrig 
			THEN //Reset error
				Error										:= FALSE;
				ErrorId										:= 0;
				ErrorFnc									:= '';	
				WinsockErrorId								:= WSOK;			
			END_IF		
		ELSIF Online
		THEN
			IF DblBuffer.ReadyToRead 			
			THEN
				CntNoOfStoredMsgs							:= 0;
				StartTimeSendMsgs							:= TIME();

				SocketUdpSend(
					sSrvNetId	:= , 
					hSocket		:= hSocket, 
					sRemoteHost	:= RemoteHost, 
					nRemotePort	:= RemotePort, 
					cbLen		:= DblBuffer.SizeOfDataToRead, 
					pSrc		:= DblBuffer.pDataToRead, 
					bExecute	:= TRUE, 
					tTimeout	:= , 
					bBusy		=> , 
					bError		=> , 
					nErrId		=> );
													
				state										:= 20;
			END_IF
		ELSIF Enable			
		THEN
			DblBuffer.SizeOfMemory							:= SizeOfBuffer;
			SocketUdpCreate(bExecute := FALSE);
			SocketClose(bExecute := FALSE);
			SocketUdpSend(bExecute := FALSE);
			Online											:= FALSE;
			Busy											:= TRUE;
			Error											:= FALSE;
			ErrorId											:= 0;
			ErrorFnc										:= '';	
			WinsockErrorId									:= WSOK;
			
			IF NOT SocketUdpCreate.bBusy
				AND NOT SocketClose.bBusy
				AND NOT SocketUdpSend.bBusy
			THEN
				state										:= 10;
			END_IF	
		ELSE //Disabled
			IF NOT DblBuffer.Empty AND Options.5
			THEN //Write rest of buffer
				IF NOT DblBuffer.ReadyToRead THEN DblBuffer.setReadyToRead(TRUE); END_IF 
				CntNoOfStoredMsgs							:= 0;
				StartTimeSendMsgs							:= TIME();
				SocketUdpSend(
					sSrvNetId	:= , 
					hSocket		:= hSocket, 
					sRemoteHost	:= RemoteHost, 
					nRemotePort	:= RemotePort, 
					cbLen		:= DblBuffer.SizeOfDataToRead, 
					pSrc		:= DblBuffer.pDataToRead, 
					bExecute	:= TRUE, 
					tTimeout	:= , 
					bBusy		=> , 
					bError		=> , 
					nErrId		=> );
				State										:= 20;
			ELSE //Close socket
				State										:= 30;
			END_IF			
		END_IF

	(* Create Socket *******************************************************)
	10: 
		SocketUdpCreate(
			sSrvNetId	:= , 
			sLocalHost	:= LocalHost, 
			nLocalPort	:= LocalPort, 
			bExecute	:= TRUE, 
			tTimeout	:= , 
			bBusy		=> , 
			bError		=> , 
			nErrId		=> , 
			hSocket		=> hSocket);
			
		IF NOT SocketUdpCreate.bBusy
		THEN
			IF SocketUdpCreate.bError
			THEN
				Error										:= TRUE;
				ErrorId										:= SocketUdpCreate.nErrId;
				ErrorFnc									:= 'SocketUdpCreate';
				WinsockErrorId								:= ADSERROR_TO_WSERROR(ErrorId);
				
				IF (Options AND OPTION_ENABLE_DEBUG) = 1
				THEN
					AdsLogError(CONCAT('LogbookClientSysLog | SocketUdpCreate %s | error id 16#', DWORD_TO_HEXSTR(TO_DWORD(ErrorID),4,FALSE)) ,HSOCKET_TO_STRING(SocketUdpCreate.hSocket));
				END_IF	

				state										:= 30;
			ELSE				
				hSocket.remoteAddr.sAddr					:= RemoteHost;
				hSocket.remoteAddr.nPort					:= RemotePort;
				
				IF (Options AND OPTION_ENABLE_DEBUG) = 1
				THEN
					AdsLogError(CONCAT('LogbookClientSysLog | SocketUdpCreate %s done', '') , HSOCKET_TO_STRING(SocketUdpCreate.hSocket));
				END_IF	
				
				Online 										:= TRUE;
				state										:= 0;
			END_IF		
			SocketUdpCreate(bExecute:= FALSE);
		END_IF		
		
	(* Send message ****************************************************)
	20:
		SocketUdpSend(
			sSrvNetId	:= , 
			hSocket		:= hSocket, 
			sRemoteHost	:= RemoteHost, 
			nRemotePort	:= RemotePort, 
			cbLen		:= DblBuffer.SizeOfDataToRead, 
			pSrc		:= DblBuffer.pDataToRead, 
			bExecute	:= TRUE, 
			tTimeout	:= , 
			bBusy		=> , 
			bError		=> , 
			nErrId		=> );
					
		IF NOT SocketUdpSend.bBusy
		THEN
			IF SocketUdpSend.bError
			THEN
				IF SendErrorCnt >= 3
				THEN
					Error									:= TRUE;
					ErrorId									:= SocketUdpSend.nErrId;
					ErrorFnc								:= 'SocketUdpSend';
					WinsockErrorId							:= ADSERROR_TO_WSERROR(ErrorId);
	
					IF (Options AND OPTION_ENABLE_DEBUG) = 1
					THEN
						AdsLogError(CONCAT('LogbookClientSysLog | SocketUdpSend %s | error id 16#', DWORD_TO_HEXSTR(TO_DWORD(ErrorID),4,FALSE)) ,HSOCKET_TO_STRING(SocketUdpCreate.hSocket));
					END_IF	
					
					State									:= 30; //Close socket
				ELSE //Try to send a second time
					SendErrorCnt							:= SendErrorCnt + 1;
				END_IF
			ELSE				
				SendErrorCnt								:= 0;	
				State										:= 0;			
			END_IF 
			DblBuffer.setReadyToRead(FALSE);
			SocketUdpSend(bExecute := FALSE);
		END_IF
		
	(* Close socket ***********************************************)
	30:	
		SocketClose(
			sSrvNetId	:= , 
			hSocket		:= SocketUdpCreate.hSocket, 
			bExecute	:= TRUE, 
			tTimeout	:= , 
			bBusy		=> , 
			bError		=> , 
			nErrId		=> );

